Yaskawa INFORM job: X2_8A-21A(90,0)_DOD_WZM_BOK.JBI

/JOB
//NAME X2_8A-21A(90,0)_DOD_WZM_BOK
///FOLDERNAME X2
//POS
///NPOS 1047,1047,1047,43,0,0
///TOOL 0
///POSTYPE PULSE
///PULSE
C00000=-12667,-135547,-130714,31270,45596,0
C00001=-9315,-159766,-119262,-3212,6219,55552
C00002=-157761,-135547,-130714,31270,45596,-69143
C00003=-154472,-113934,-104337,41712,51336,-70449
C00004=-149832,-108771,-100172,39130,49259,-68869
C00005=-148058,-106656,-98467,38074,48499,-68236
C00006=-148062,-106275,-96666,38578,47777,-68578
C00007=-148058,-106656,-98467,38074,48499,-68236
C00008=-147997,-106381,-96958,38469,47847,-68508
C00009=-145894,-104035,-96109,36815,47477,-67498
C00010=-147997,-106381,-96958,38469,47847,-68508
C00011=-154410,-113635,-102825,42095,50721,-70729
C00012=-154342,-120637,-107041,25827,48602,-38771
C00013=-150292,-111683,-102360,22573,48994,-36710
C00014=-148798,-108210,-100464,21373,49171,-35962
C00015=-146664,-105787,-99597,19708,49308,-34937
C00016=-146949,-106220,-99797,19932,49282,-35074
C00017=-147721,-103636,-97533,20478,49410,-35405
C00018=-146949,-106220,-99797,19932,49282,-35074
C00019=-152261,-118724,-106469,24248,48548,-37770
C00020=-148295,-114597,-117137,-6490,60568,-69086
C00021=-147868,-109631,-111600,-6790,59752,-68875
C00022=-147704,-107727,-109395,-6911,59390,-68790
C00023=-147708,-107860,-107783,-6984,58336,-68724
C00024=-147704,-107727,-109395,-6911,59390,-68790
C00025=-147723,-107760,-107968,-6963,58499,-68740
C00026=-147306,-102596,-106094,-7098,60024,-68678
C00027=-147723,-107760,-107968,-6963,58499,-68740
C00028=-148315,-114751,-115749,-6537,59639,-69038
C00029=-148355,-114889,-117236,-6461,60467,-69101
C00030=-147925,-109892,-111692,-6763,59663,-68890
C00031=-147761,-107977,-109485,-6884,59305,-68805
C00032=-147764,-108104,-107870,-6957,58254,-68739
C00033=-147777,-108153,-108078,-6942,58354,-68751
C00034=-147358,-102980,-106206,-7078,59886,-68688
C00035=-147777,-108153,-108078,-6942,58354,-68751
C00036=-148373,-115211,-115873,-6515,59468,-69049
C00037=-147696,-122269,-111871,-35505,39043,-51945
C00038=-147690,-118447,-100224,-39719,34874,-49579
C00039=-148491,-109409,-94254,-38171,35277,-50420
C00040=-148787,-105724,-91002,-38010,35060,-50504
C00041=-148789,-105382,-89977,-38411,34697,-50285
C00042=-149058,-101689,-89016,-37046,35623,-51030
C00043=-149145,-100783,-88679,-36755,35795,-51189
C00044=-149058,-101689,-89016,-37046,35623,-51030
C00045=-145777,-99657,-88811,-39022,37803,-49998
C00046=-148139,-100407,-89095,-37251,36591,-50936
C00047=-145777,-99657,-88811,-39022,37803,-49998
C00048=-147690,-118447,-100224,-39719,34874,-49579
C00049=-128033,-128545,-103748,-39689,32513,-43973
C00050=-128383,-118409,-97778,-37905,33566,-44930
C00051=-128511,-114277,-94563,-37658,33626,-45064
C00052=-128512,-113804,-93446,-38069,33271,-44843
C00053=-129119,-111006,-93029,-36452,33958,-45715
C00054=-129434,-109852,-92636,-35862,34111,-46033
C00055=-128358,-113721,-93936,-37885,33613,-44941
C00056=-176216,-70111,-78093,55162,70856,-80763
C00057=-174311,-70781,-78417,54616,69674,-80426
C00058=-176216,-70111,-78093,55162,70856,-80763
C00059=-181747,-69996,-81392,56304,75271,-81045
C00060=-178033,-77165,-93769,42680,75059,-77098
C00061=-164745,-109340,-116699,-3009,62053,-68278
C00062=-145851,-112599,-102075,-47717,41998,-56322
C00063=-148044,-104803,-96379,-45883,41204,-57334
C00064=-148864,-101708,-93474,-45490,40644,-57533
C00065=-148866,-101457,-92299,-45986,40221,-57239
C00066=-148863,-101834,-94104,-45225,40876,-57690
C00067=-145127,-99228,-91361,-47944,42572,-56214
C00068=-147466,-100038,-91670,-46636,41186,-56907
C00069=-145127,-99228,-91361,-47944,42572,-56214
C00070=-146129,-107372,-95667,-48598,40993,-55782
C00071=-148216,-109089,-93488,-49289,38371,-55335
C00072=-148344,-107837,-93052,-48851,38553,-55585
C00073=-147906,-112054,-94498,-50363,37947,-54724
C00074=-145851,-112599,-102075,-47717,41998,-56322
C00075=-158250,-140903,-124067,-47621,67451,-49320
C00076=-161740,-133075,-117656,-46661,65672,-50232
C00077=-162335,-130592,-114553,-46699,64919,-50156
C00078=-162276,-129951,-113381,-46845,64676,-49998
C00079=-160420,-132544,-115533,-47350,65644,-49520
C00080=-135901,-74424,-73697,-74364,100921,-31256
C00081=-137788,-75503,-74147,-74218,99532,-31324
C00082=-138769,-76027,-74362,-74146,98812,-31363
C00083=-135901,-74424,-73697,-74364,100921,-31256
C00084=-149282,-147643,-98518,-79858,51263,-26133
C00085=-149394,-146891,-98381,-79629,51249,-26315
C00086=-148448,-152811,-99407,-81432,51428,-24854
C00087=-139735,-166147,-105854,-82069,56849,-22658
C00088=-180438,-97574,-115199,-33764,102267,52414
C00089=-189965,-108899,-115705,-31971,94091,51156
C00090=-190633,-110068,-115194,-31831,93066,51189
C00091=-190637,-110288,-114404,-31804,92551,51332
C00092=-190629,-109833,-115910,-31859,93547,51055
C00093=-186867,-102382,-113240,-32521,96788,51574
C00094=-187005,-102964,-110979,-32373,95300,51952
C00095=-188888,-106610,-112304,-32065,93703,51681
C00096=-187005,-102964,-110979,-32373,95300,51952
C00097=-188021,-107681,-112675,-32159,93748,52003
C00098=-189590,-103281,-111094,-32025,94271,51250
C00099=-188021,-107681,-112675,-32159,93748,52003
C00100=-180438,-97574,-115199,-33764,102267,52414
C00101=-185735,-83978,-109774,-33564,103394,50026
C00102=-199988,-77820,-108712,11582,98175,-38155
C00103=-204749,-56978,-92496,29836,109182,-47433
C00104=-202460,-56662,-91339,29422,107990,-46925
C00105=-201413,-57385,-91726,29256,107546,-46663
C00106=-201611,-57041,-91542,29296,107663,-46703
C00107=-201611,-58240,-90431,29070,106521,-47008
C00108=-203359,-50274,-87822,29763,109247,-46906
C00109=-195470,-25798,-72981,29209,109868,-43903
C00110=-195013,-27562,-73704,29036,109327,-43888
C00111=-194283,-28250,-74172,28893,109053,-43704
C00112=-194480,-28066,-74047,28932,109127,-43754
C00113=-194480,-29296,-73135,28708,108075,-44034
C00114=-195605,-24849,-71507,29147,109538,-44038
C00115=-191110,-5546,-57842,28597,109561,-42465
C00116=-192519,-3768,-54500,33008,111368,-41387
C00117=-191992,-5303,-55742,32912,111174,-41254
C00118=-192059,-5108,-55586,32924,111198,-41271
C00119=-192059,-6294,-54683,32651,110210,-41583
C00120=-192882,-2296,-53893,33162,111810,-41382
C00121=-203365,-15491,-64400,34648,115083,-44256
C00122=-218411,-26661,-75493,58573,107247,-46176
C00123=-145332,-87800,-123084,4045,108310,15756
C00124=-109199,-104290,-129101,-21867,105305,43874
C00125=-112610,-115777,-129409,-14908,94573,36374
C00126=-117115,-112620,-124614,-14006,92529,35127
C00127=-118008,-112320,-123068,-13816,91609,34934
C00128=-118007,-112900,-122267,-13806,90840,35020
C00129=-118044,-112536,-122505,-13803,91159,34973
C00130=-118576,-105776,-120168,-13731,93052,34586
C00131=-118044,-112536,-122505,-13803,91159,34973
C00132=-125955,-111499,-122045,-12179,90192,32457
C00133=-127333,-111877,-122174,-11884,89885,32033
C00134=-124755,-111115,-121914,-12435,90480,32824
C00135=-119624,-116552,-128230,-13509,92325,34321
C00136=-117231,-121833,-124467,-22052,85463,28755
C00137=-122341,-114124,-118662,-20866,84531,27121
C00138=-123318,-113111,-117155,-20643,83910,26885
C00139=-123641,-113323,-116249,-20585,83205,26892
C00140=-123595,-112804,-116375,-20585,83540,26851
C00141=-123397,-106736,-114247,-20589,85286,26623
C00142=-123595,-112804,-116375,-20585,83540,26851
C00143=-116023,-114044,-115764,-22346,84523,29358
C00144=-117346,-116777,-115957,-22098,82979,29171
C00145=-118867,-116723,-116143,-21757,82713,28674
C00146=-116293,-116772,-115815,-22329,83179,29512
C00147=-117231,-121833,-124467,-22052,85463,28755
C00148=-154726,-134692,-133300,19029,79240,32627
C00149=-155157,-123239,-125350,19102,80279,32639
C00150=-155214,-122106,-123677,19140,79867,32554
C00151=-155216,-122330,-122794,19175,79245,32454
C00152=-155272,-122641,-123186,19186,79334,32449
C00153=-154565,-115790,-120970,18882,81218,32994
C00154=-155272,-122449,-123985,19155,79894,32538
C00155=-110972,-119209,-121408,-15853,79302,48266
C00156=-109086,-133769,-122042,-16854,72857,49812
C00157=-111848,-135958,-122676,-16103,71595,48979
C00158=-109086,-133769,-122042,-16854,72857,49812
C00159=-108592,-130707,-130810,-16554,79646,49045
C00160=-120610,-122471,-119242,-21572,81234,22537
C00161=-120610,-122484,-118172,-21604,80613,22649
C00162=-120610,-122391,-116483,-21658,79689,22817
C00163=-120610,-122419,-116833,-21647,79876,22783
C00164=-120610,-122423,-116832,-21647,79874,22783
C00165=-120610,-122419,-116833,-21647,79876,22783
C00166=-120610,-122416,-116761,-21649,79836,22790
C00167=-120610,-122436,-116768,-21650,79830,22791
C00168=-120610,-122416,-116761,-21649,79836,22790
C00169=-120611,-122370,-120508,-21535,82009,22397
C00170=-120500,-119354,-126515,-17332,87675,17755
C00171=-155157,-123239,-125350,19102,80279,32639
C00172=-155214,-122106,-123677,19140,79867,32554
C00173=-155216,-122330,-122794,19175,79245,32454
C00174=-155272,-122641,-123186,19186,79334,32449
C00175=-154565,-115790,-120970,18882,81218,32994
C00176=-155272,-122449,-123985,19155,79894,32538
C00177=-110972,-119209,-121408,-15853,79302,48266
C00178=-109086,-133769,-122042,-16854,72857,49812
C00179=-111848,-135958,-122676,-16103,71595,48979
C00180=-109086,-133769,-122042,-16854,72857,49812
C00181=-108592,-130707,-130810,-16554,79646,49045
C00182=-120611,-118687,-129075,-3134,90000,4412
C00183=-120611,-121772,-123926,-3138,85252,4531
C00184=-120611,-122092,-122744,-3141,84362,4553
C00185=-120611,-122362,-121169,-3146,83256,4581
C00186=-120611,-122286,-121724,-3144,83636,4571
C00187=-120611,-122290,-121724,-3144,83633,4571
C00188=-120611,-122286,-121724,-3144,83636,4571
C00189=-120611,-121006,-125813,-3134,86805,4492
C00190=-120621,-113915,-131911,-13153,116790,34478
C00191=-136832,-143297,-133894,-19017,104291,40845
C00192=-187686,-122249,-118318,-34521,102174,42234
C00193=-187703,-122088,-115580,-34298,100833,42653
C00194=-187707,-122010,-114917,-34250,100525,42749
C00195=-187713,-121734,-113169,-34135,99743,42991
C00196=-187707,-122010,-114917,-34250,100525,42749
C00197=-187770,-121697,-112491,-32279,113674,44764
C00198=-187767,-121692,-112491,-32279,113678,44765
C00199=-187770,-121697,-112491,-32279,113674,44764
C00200=-187667,-121438,-112064,-34928,84963,41689
C00201=-187673,-121448,-112068,-34927,84958,41688
C00202=-187667,-121438,-112064,-34928,84963,41689
C00203=-187641,-121360,-124129,-34919,91154,39753
C00204=-178673,-119471,-127738,-23493,103847,53429
C00205=-160878,-120510,-126471,-37,121976,81968
C00206=-160881,-121699,-123664,-37,119637,81967
C00207=-160883,-121991,-122485,-37,118762,81967
C00208=-160886,-122244,-120905,-37,117660,81966
C00209=-160884,-122111,-121864,-37,118318,81967
C00210=-160882,-122100,-121862,-36,118322,81968
C00211=-160884,-122111,-121864,-37,118318,81967
C00212=-160879,-120821,-125908,-37,121469,81968
C00213=-160879,-120821,-131564,-37,121469,81968
C00214=-157394,-128671,-131753,738,117538,83283
C00215=-158801,-138021,-132727,409,113343,82737
C00216=-158801,-138035,-132347,409,113101,82737
C00217=-158801,-138034,-131509,408,112586,82736
C00218=-158801,-138039,-131833,408,112783,82736
C00219=-160693,-149427,-134985,6,108877,82039
C00220=-160612,-153549,-136083,24,107435,82069
C00221=-159125,-144348,-133603,336,110634,82611
C00222=-199963,-104116,-119881,11013,127404,83152
C00223=-204692,-116225,-118816,8637,121169,80600
C00224=-203581,-121519,-120530,8810,119404,80895
C00225=-204849,-113790,-122122,8953,124435,80816
C00226=-166129,-114439,-129167,13521,133132,-54375
C00227=-82387,-124374,-130385,21792,102809,-55833
C00228=-37550,-124758,-124791,27166,84975,-54517
C00229=-35933,-124831,-122904,26864,83389,-54284
C00230=-35589,-124875,-121597,26827,82538,-54351
C00231=-35584,-124889,-121174,26839,82296,-54405
C00232=-35764,-126387,-121953,26892,82093,-54519
C00233=-31633,-125451,-121673,25972,81076,-53208
C00234=-35764,-126387,-121953,26892,82093,-54519
C00235=-46981,-157328,-126723,35790,81436,-33730
C00236=-42905,-153934,-122174,35701,78867,-32870
C00237=-42758,-143813,-119569,35389,81762,-31868
C00238=-42905,-153934,-122174,35701,78867,-32870
C00239=-53188,-117519,-120731,36414,97747,-30962
C00240=-95179,-109851,-129540,3422,106316,17944
C00241=-143691,-100776,-119079,-26047,122130,73021
C00242=-146029,-112499,-120098,-24937,116556,73463
C00243=-147204,-116618,-119576,-24569,113992,73590
C00244=-147487,-116577,-118677,-24502,113425,73607
C00245=-146967,-116625,-120319,-24630,114475,73574
C00246=-147345,-121113,-121824,-24401,113105,73737
C00247=-146899,-128254,-123879,-23878,111030,74376
C00248=-147345,-121113,-121824,-24401,113105,73737
C00249=-118081,-135478,-120686,-30293,109901,65237
C00250=-118366,-136707,-118609,-29972,108136,65614
C00251=-120887,-140213,-119894,-30302,106351,65070
C00252=-118366,-136707,-118609,-29972,108136,65614
C00253=-117820,-130449,-123242,-31209,113594,64262
C00254=-93926,-103398,-125362,-18301,106221,39936
C00255=-72688,-110808,-124077,-7134,85250,24096
C00256=-75848,-101444,-116923,-6191,85411,23073
C00257=-76170,-100985,-115528,-6097,84767,23002
C00258=-76167,-101481,-114835,-6104,84090,23035
C00259=-78739,-96930,-113773,-5320,85595,22140
C00260=-79843,-95445,-113201,-4985,85938,21775
C00261=-77748,-98228,-114268,-5620,85298,22470
C00262=-140085,-104632,-109249,40944,98797,-6712
C00263=-140263,-103640,-106572,40817,98007,-7102
C00264=-137942,-102173,-106029,40697,97269,-6378
C00265=-140263,-103640,-106572,40817,98007,-7102
C00266=-135988,-101428,-112112,41019,99549,-4631
C00267=-141957,-83285,-117139,12315,91699,6710
C00268=-161957,-129781,-122866,-20018,67926,12328
C00269=-166016,-109699,-113650,-17211,72980,10098
C00270=-166795,-105246,-111748,-16434,74862,9605
C00271=-165677,-113012,-111900,-18316,68836,10778
C00272=-162725,-116093,-113629,-19548,69016,11850
C00273=-162651,-107484,-110669,-19284,71494,11460
C00274=-162725,-116093,-113629,-19548,69016,11850
C00275=-155151,-112727,-112486,-22270,71877,14160
C00276=-155120,-113819,-110277,-22518,70103,14518
C00277=-159000,-114269,-110433,-21107,68960,13264
C00278=-155120,-113819,-110277,-22518,70103,14518
C00279=-155137,-138999,-124748,-23105,66364,15269
C00280=-81055,-115973,-127517,23586,109336,-64560
C00281=-76492,-127739,-126040,22738,101683,-64421
C00282=-76072,-128597,-125529,22671,100870,-64425
C00283=-76065,-128640,-125326,22657,100732,-64448
C00284=-76072,-128576,-125785,22685,101025,-64394
C00285=-82641,-146978,-130130,22016,96499,-67668
C00286=-81130,-155003,-132256,21951,93476,-67670
C00287=-82641,-146978,-130130,22016,96499,-67668
C00288=-84000,-144678,-127518,21929,96467,-68175
C00289=-84000,-143983,-126065,21900,95967,-68269
C00290=-83327,-146231,-127404,21916,95478,-68108
C00291=-88356,-135439,-132684,22407,104994,-68175
C00292=-104080,-128245,-132212,-31995,84146,-22143
C00293=-106783,-105266,-117364,-31197,85468,-23533
C00294=-107129,-103609,-115494,-31111,85090,-23558
C00295=-107127,-104217,-114421,-31144,84251,-23329
C00296=-107044,-104571,-114816,-31164,84333,-23320
C00297=-107880,-99055,-112779,-30885,85404,-23924
C00298=-107044,-104571,-114816,-31164,84333,-23320
C00299=-105114,-115284,-123193,-31689,84721,-22698
C00300=-105208,-113465,-123990,-31624,85910,-23065
C00301=-106823,-104635,-117017,-31184,85549,-23570
C00302=-107122,-103295,-115264,-31113,85109,-23561
C00303=-107121,-103855,-114286,-31142,84342,-23351
C00304=-107087,-104437,-114776,-31151,84356,-23343
C00305=-107921,-98925,-112738,-30873,85426,-23945
C00306=-107087,-104437,-114776,-31151,84356,-23343
C00307=-105701,-116384,-125830,-31502,85418,-23114
C00308=-79137,-116524,-127291,-7118,77084,38210
C00309=-66518,-158449,-133200,-8588,59166,50817
C00310=-70166,-147728,-127011,-6864,60501,49298
C00311=-71549,-143558,-123868,-6244,60595,48757
C00312=-71544,-142942,-122687,-6271,60188,48782
C00313=-71412,-140542,-122600,-6259,61371,48766
C00314=-74130,-137647,-121783,-5023,62161,47690
C00315=-71412,-140542,-122600,-6259,61371,48766
C00316=-59221,-85077,-106862,-19044,97138,55247
C00317=-59772,-90133,-108950,-18878,95774,55276
C00318=-59221,-85077,-106862,-19044,97138,55247
C00319=-65406,-128676,-128270,-8670,80773,42177
C00320=-57064,-112054,-129147,-2862,108793,29097
C00321=-70948,-123089,-127271,10962,111372,-380
C00322=-67644,-116564,-123033,11394,111660,848
C00323=-67644,-116773,-122597,11361,111292,811
C00324=-67644,-116291,-123546,11437,112109,893
C00325=-70770,-123262,-125779,10903,110357,-412
C00326=-70770,-123588,-124717,10837,109552,-488
C00327=-69306,-120453,-123728,11077,110342,115
C00328=-70770,-123283,-125719,10898,110311,-416
C00329=-70770,-119886,-130778,11344,115083,53
C00330=-68413,-122856,-123349,22437,117236,58
C00331=-67404,-122631,-120786,22344,115611,123
C00332=-67401,-122683,-120099,22253,115193,37
C00333=-67283,-122594,-120333,22317,115338,115
C00334=-65261,-118175,-118917,23034,116088,1096
C00335=-67283,-122594,-120333,22317,115338,115
C00336=-70820,-123560,-126018,22187,119059,-540
C00337=-59587,-128850,-129971,-18356,103459,48793
C00338=-60648,-112549,-116046,-37363,97913,74718
C00339=-66648,-121539,-115269,-36526,91263,74498
C00340=-69624,-125916,-115212,-36242,88151,74300
C00341=-69624,-125773,-114639,-36242,87924,74374
C00342=-69624,-125814,-114800,-36242,87987,74354
C00343=-70738,-127677,-115368,-36152,87024,74211
C00344=-69624,-125814,-114800,-36242,87987,74354
C00345=-61556,-115340,-115782,-37136,96245,74919
C00346=-93863,-107857,-129738,-18786,98098,27923
C00347=-113340,-105978,-120535,-17383,92037,15860
C00348=-116256,-99504,-115214,-16745,91512,14962
C00349=-117355,-97038,-113094,-16498,91266,14630
C00350=-124053,-106600,-116618,-14934,87391,12894
C00351=-123019,-109757,-118902,-15179,87365,13243
C00352=-120254,-118381,-124729,-15823,87055,14212
C00353=-121076,-118719,-112405,-41381,81563,9211
C00354=-125328,-110839,-107644,-40465,80446,7775
C00355=-126920,-107772,-105722,-40091,80023,7243
C00356=-122279,-105715,-102241,-45382,81605,7865
C00357=-118123,-103314,-98388,-50429,83325,8212
C00358=-115452,-99808,-95169,-50805,84680,8860
C00359=-113598,-101964,-96694,-51043,85596,9323
C00360=-108732,-107177,-100380,-51565,88044,10518
C00361=-131658,-113091,-133069,-11905,90618,-13395
C00362=-155934,-143784,-122811,23124,58745,-32427
C00363=-151507,-132468,-117411,20635,59886,-30339
C00364=-149876,-128251,-115276,19729,60288,-29596
C00365=-151213,-128323,-114307,20456,60014,-30191
C00366=-146890,-120795,-114089,13688,65901,-25886
C00367=-142734,-111238,-112703,7950,73001,-22079
C00368=-143750,-114926,-115045,8343,72653,-22456
C00369=-146492,-125018,-121022,9420,71459,-23506
C00370=-146459,-122334,-129315,9145,77857,-23007
C00371=-118526,-115013,-133262,8809,105739,-46794
C00372=-93674,-118800,-129721,8134,120991,-68616
C00373=-93669,-120967,-127104,7892,118292,-68817
C00374=-94734,-125499,-127256,7488,116172,-69370
C00375=-102152,-150969,-134401,5465,108121,-72564
C00376=-93660,-121042,-127131,7893,118270,-68815
C00377=-93665,-118880,-129750,8134,120967,-68614
C00378=-98446,-113408,-116165,41475,93741,-73013
C00379=-95217,-118830,-115137,40946,89638,-73223
C00380=-92912,-120932,-114950,40678,87660,-72983
C00381=-96081,-129446,-114840,41081,85733,-75123
C00382=-96936,-125131,-114749,41104,87782,-74702
C00383=-101504,-121000,-116278,41571,92256,-74948
C00384=-100864,-122088,-112493,43204,76282,-71688
C00385=-96953,-122826,-110054,42689,72984,-71279
C00386=-94356,-123741,-109617,42253,71173,-70830
C00387=-94321,-123299,-107872,42432,70522,-71095
C00388=-95642,-121622,-108630,42447,72155,-71017
C00389=-100864,-121830,-111367,43291,75868,-71867
C00390=-131033,-115476,-133015,2815,101744,-74384
C00391=-151471,-119125,-123137,-34971,103386,-73225
C00392=-162012,-101235,-114016,-37763,108592,-75954
C00393=-165544,-104560,-113885,-37278,105688,-76399
C00394=-161186,-105898,-111701,-36934,105869,-74609
C00395=-157962,-101866,-111865,-37402,108959,-74341
C00396=-155898,-93647,-112180,-38609,113341,-75115
C00397=-93674,-112333,-133466,8753,126560,-68151
C00398=-93674,-118800,-129721,8134,120991,-68616
C00399=-93669,-120967,-127104,7892,118292,-68817
C00400=-93667,-121558,-126026,7814,117333,-68886
C00401=-93663,-121536,-126144,7822,117416,-68879
C00402=-93639,-121762,-126135,7818,117296,-68878
C00403=-93680,-121434,-126040,7817,117406,-68885
C00404=-93660,-121042,-127131,7893,118270,-68815
C00405=-93665,-118880,-129750,8134,120967,-68614
C00406=-98446,-113408,-116165,41475,93741,-73013
C00407=-93996,-117843,-114815,40802,89312,-72817
C00408=-91343,-117266,-113836,40455,87860,-72224
C00409=-92137,-119395,-114109,40564,87510,-72703
C00410=-95072,-126184,-113786,40951,86041,-74561
C00411=-95071,-125918,-112907,40977,85731,-74679
C00412=-96936,-125131,-114749,41104,87782,-74702
C00413=-101504,-121000,-116278,41571,92256,-74948
C00414=-100864,-122088,-112493,43204,76282,-71688
C00415=-95643,-121963,-109784,42340,72556,-70846
C00416=-93677,-120964,-108398,41948,71358,-70433
C00417=-93599,-120925,-107098,42100,70733,-70661
C00418=-95642,-121622,-108630,42447,72155,-71017
C00419=-100864,-121830,-111367,43291,75868,-71867
C00420=-131033,-115476,-133015,2815,101744,-74384
C00421=-151471,-119125,-123137,-34971,103386,-73225
C00422=-162012,-101235,-114016,-37763,108592,-75954
C00423=-163593,-104354,-113811,-37340,106547,-75879
C00424=-162938,-104376,-113793,-37349,106803,-75692
C00425=-158829,-104862,-111593,-37019,107224,-74083
C00426=-157962,-101866,-111865,-37402,108959,-74341
C00427=-155898,-93647,-112180,-38609,113341,-75115
C00428=-179206,-139250,-107986,-62075,77828,-66561
C00429=-185232,-138953,-105140,-62379,73225,-66913
C00430=-187696,-139015,-104542,-62453,71468,-67163
C00431=-187702,-137665,-102648,-62587,71237,-66963
C00432=-185238,-138055,-103864,-62461,73065,-66778
C00433=-179211,-138396,-106727,-62132,77661,-66424
C00434=-179188,-148562,-121526,-61524,79591,-68010
C00435=-184417,-115822,-131978,-19629,107310,7500
C00436=-190427,-134899,-136820,8574,116374,78562
C00437=-188066,-120573,-128029,9218,118052,79593
C00438=-191610,-147357,-136376,6897,103791,75181
C00439=-187795,-119828,-126345,9210,117376,79639
C00440=-187841,-121664,-124728,-2971,114560,78170
C00441=-187942,-121398,-126015,-3016,115485,78109
C00442=-187937,-119495,-128851,-3098,118205,78035
C00443=-176042,-128909,-129640,-7380,110692,58022
C00444=-187833,-113452,-115854,-34994,105139,41767
C00445=-187847,-113781,-113588,-34722,103839,42187
C00446=-187853,-113844,-112659,-34623,103335,42348
C00447=-187856,-113866,-111596,-34519,102780,42525
C00448=-187851,-113844,-112538,-34611,103274,42368
C00449=-187836,-113627,-114840,-34866,104547,41960
C00450=-186756,-108501,-120882,-36201,110201,40487
C00451=-150585,-129060,-123753,-46684,114085,-39870
C00452=-134046,-137019,-115206,-49635,112096,-74674
C00453=-134033,-140586,-110307,-48065,108843,-72866
C00454=-134037,-138671,-107458,-47843,108316,-72589
C00455=-133950,-137111,-106105,-47812,108341,-72556
C00456=-133930,-150358,-126108,1173,113974,-57522
C00457=-134040,-150029,-126001,1133,114079,-57562
C00458=-134505,-148512,-125722,2741,114238,-57140
C00459=-137673,-151162,-132623,1623,117206,-58299
C00460=-106012,-107394,-121753,14018,130776,-44816
C00461=-106669,-102485,-112824,13121,127987,-45519
C00462=-97512,-96218,-110425,14566,129183,-82759
C00463=-98864,-105619,-112306,13303,125832,-83842
C00464=-106150,-109468,-113796,12766,125107,-45727
C00465=-105474,-116823,-114648,29161,97726,-33837
C00466=-134074,-146851,-118858,40485,90771,-46834
C00467=-141855,-151854,-132376,33568,89282,-32323
C00468=-173958,-148748,-133240,11874,65312,15203
C00469=-187653,-128002,-123664,-7056,57779,46476
C00470=-188071,-112180,-99768,1790,31671,46486
C00471=-188092,-111455,-97340,1875,30550,46442
C00472=-187851,-111485,-96835,1581,30220,46589
C00473=-187792,-110201,-93997,1555,29133,46605
C00474=-187737,-110060,-93474,1490,28882,46636
C00475=-187785,-109075,-90961,1604,27844,46576
C00476=-188106,-109627,-92159,2030,28303,46362
C00477=-188086,-110531,-94662,1935,29378,46411
C00478=-188086,-114129,-114927,1479,39995,46659
C00479=-201470,-41376,-102585,19941,97743,-57993
C00480=-197439,-2624,-49840,39121,107911,-51008
C00481=-168348,92819,48556,27514,116832,-48709
C00482=-170146,82769,36005,28011,119675,-48673
C00483=-172466,59662,8523,30747,114377,-38085
C00484=-173361,44293,-8668,31536,116980,-37634
C00485=-173326,42548,-10417,31798,119739,-39927
C00486=-173293,31446,-22173,31559,124382,-42741
C00487=-170045,43132,-9775,28753,130915,-51393
C00488=-186843,33187,-28183,45340,118495,-56566
C00489=-187270,22965,-40018,42118,113549,-44205
C00490=-164927,12374,-50848,37497,97302,26684
C00491=-160848,-52651,-98971,6904,73590,44156
C00492=-187933,-111679,-98706,-278,30585,46526
C00493=-187953,-110958,-96368,-260,29517,46517
C00494=-188171,-110591,-95666,34,29272,46369
C00495=-188111,-109885,-93130,-50,28074,46412
C00496=-188090,-109778,-92606,-82,27808,46427
C00497=-188055,-108797,-90194,-133,26826,46455
C00498=-187968,-109087,-91174,-258,27282,46516
C00499=-187948,-109974,-93584,-278,28309,46526
C00500=-190713,-138118,-122139,3147,45685,54861
C00501=-188097,-104568,-127563,3199,90457,72619
C00502=-188112,-108983,-124849,3203,86524,72515
C00503=-196049,-130715,-128058,11352,73875,69900
C00504=-193131,-119078,-125609,7963,80164,71095
C00505=-187364,-124777,-127140,2732,76642,72458
C00506=-191510,-130298,-128202,6704,73471,71168
C00507=-188153,-109076,-124888,3215,86502,72501
C00508=-188138,-104664,-127604,3212,90434,72606
C00509=-187898,-111965,-120493,-16766,69565,69566
C00510=-187918,-113285,-117348,-17044,67055,69927
C00511=-188336,-115132,-116370,-17036,65483,70009
C00512=-188181,-112945,-115606,-17029,66143,69965
C00513=-188166,-113080,-115592,-17048,66072,69982
C00514=-187991,-112297,-115306,-17102,66325,70009
C00515=-187944,-113344,-117352,-17035,67023,69922
C00516=-187924,-112030,-120500,-16757,69531,69561
C00517=-180038,-109975,-126789,-2440,82512,-7441
C00518=-174468,-102021,-118148,-1871,82653,-17547
C00519=-174479,-103807,-115834,-1877,80312,-17516
C00520=-175021,-104384,-114967,-1695,79470,-17680
C00521=-174783,-104250,-115053,-1777,79597,-17606
C00522=-174170,-106690,-109656,-11758,69864,-18312
C00523=-172833,-107431,-109671,-12341,69693,-17819
C00524=-174390,-105691,-110273,-11607,70709,-18474
C00525=-174377,-104937,-112785,-11492,72607,-18653
C00526=-190845,-100837,-124447,13698,93294,-33124
C00527=-206306,-116062,-120388,37359,88631,-50073
C00528=-215039,-120395,-106715,50971,83253,-62053
C00529=-215038,-119729,-104733,51036,82687,-62365
C00530=-215037,-119445,-103934,51064,82464,-62488
C00531=-215047,-118488,-101366,51160,81769,-62880
C00532=-215047,-118800,-102176,51129,81987,-62759
C00533=-215049,-119543,-104187,51057,82539,-62453
C00534=-215012,-122438,-115563,50746,86080,-60488
C00535=-160845,-113405,-113287,47121,77099,31472
C00536=-160851,-113463,-110064,47446,75709,30781
C00537=-161282,-114943,-109409,47754,75135,30277
C00538=-161254,-114846,-109376,47745,75139,30294
C00539=-160788,-113231,-109982,47419,75724,30819
C00540=-160782,-112987,-114684,46949,77813,31850
C00541=-161690,-87231,-108001,36248,90547,80444
C00542=-156210,-91223,-102127,34873,83736,80390
C00543=-152348,-73560,-94415,33644,85868,82536
C00544=-158330,-83683,-104653,35339,89043,81248
C00545=-160758,-112853,-114863,36163,82877,78288
C00546=-160760,-113152,-111426,36317,81029,77674
C00547=-159491,-108015,-113138,31549,97627,78488
C00548=-160662,-113202,-114930,31505,96709,77777
C00549=-163626,-124672,-119545,29271,98661,76908
C00550=-164622,-129006,-121133,28240,99357,76613
C00551=-160757,-112482,-116558,30024,102576,77779
C00552=-160755,-111254,-119690,30396,104801,78387
C00553=-139139,-104942,-132434,5076,105021,81413
C00554=-120610,-140892,-128239,-26796,83300,73925
C00555=-124485,-139346,-124335,-26282,80622,73071
C00556=-128794,-174695,-130569,-28116,58521,76693
C00557=-123854,-173705,-127920,-33486,56775,79744
C00558=-127596,-155142,-123084,-28725,56836,77726
C00559=-128095,-155529,-122172,-29132,53686,78388
C00560=-128860,-155984,-126780,-25446,58633,74277
C00561=-138109,-135032,-133743,-8289,74304,51513
C00562=-203654,-125968,-124215,37381,73551,-30645
C00563=-201127,-103516,-110680,20461,62884,-59060
C00564=-201138,-104157,-107983,20829,61019,-59420
C00565=-201193,-104400,-106652,21043,60147,-59612
C00566=-201232,-104446,-106694,21063,60161,-59627
C00567=-200873,-105228,-106882,20926,59802,-59552
C00568=-201116,-104130,-107973,20816,61021,-59411
C00569=-201105,-103488,-110669,20449,62886,-59051
C00570=-198523,-119273,-121454,24683,77158,-64296
C00571=-174403,-100049,-121231,21877,99309,-62114
C00572=-174406,-102879,-118773,21681,96545,-62622
C00573=-172958,-103152,-117900,21399,95556,-62302
C00574=-174224,-104881,-115910,21520,93897,-63036
C00575=-174418,-104205,-117181,21599,94999,-62906
C00576=-174415,-101880,-119808,21752,97619,-62429
C00577=-185776,-93152,-118465,-1785,83350,-67432
C00578=-169060,-142396,-123848,-37084,49654,-60484
C00579=-174230,-113472,-108308,-34615,49911,-64397
C00580=-174247,-112967,-104740,-35556,48304,-63744
C00581=-174471,-112928,-103062,-35946,47380,-63468
C00582=-174489,-112275,-102294,-36008,47261,-63425
C00583=-174590,-112153,-101603,-36140,46922,-63333
C00584=-174396,-113097,-100663,-36857,46141,-62871
C00585=-174330,-114043,-100633,-37190,45762,-62656
C00586=-174129,-122060,-98220,-45554,37107,-60115
C00587=-174246,-112406,-102200,-36228,47262,-63291
C00588=-174229,-113129,-105847,-35265,48804,-63944
C00589=-182962,-136134,-123657,-29797,44727,-67038
C00590=-203654,-125968,-124215,37381,73551,-30645
C00591=-201127,-103516,-110680,20461,62884,-59060
C00592=-201138,-104157,-107983,20829,61019,-59420
C00593=-201193,-104400,-106652,21043,60147,-59612
C00594=-201232,-104446,-106694,21063,60161,-59627
C00595=-200873,-105228,-106882,20926,59802,-59552
C00596=-201116,-104130,-107973,20816,61021,-59411
C00597=-201105,-103488,-110669,20449,62886,-59051
C00598=-198523,-119273,-121454,24683,77158,-64296
C00599=-174403,-100049,-121231,21877,99309,-62114
C00600=-174406,-102879,-118773,21681,96545,-62622
C00601=-172958,-103152,-117900,21399,95556,-62302
C00602=-174224,-104881,-115910,21520,93897,-63036
C00603=-174418,-104205,-117181,21599,94999,-62906
C00604=-174415,-101880,-119808,21752,97619,-62429
C00605=-185776,-93152,-118465,-1785,83350,-67432
C00606=-169060,-142396,-123848,-37084,49654,-60484
C00607=-174230,-113472,-108308,-34615,49911,-64397
C00608=-174247,-112967,-104740,-35556,48304,-63744
C00609=-174471,-112928,-103062,-35946,47380,-63468
C00610=-174489,-112275,-102294,-36008,47261,-63425
C00611=-174590,-112153,-101603,-36140,46922,-63333
C00612=-174396,-113097,-100663,-36857,46141,-62871
C00613=-174330,-114043,-100633,-37190,45762,-62656
C00614=-174129,-122060,-98220,-45554,37107,-60115
C00615=-174246,-112406,-102200,-36228,47262,-63291
C00616=-175798,-117006,-109100,-34199,48210,-64559
C00617=-178617,-124532,-114828,-32467,46840,-65534
C00618=-210827,-121899,-127370,-35396,86436,-76908
C00619=-214505,-124636,-123608,-35577,86411,-76994
C00620=-214521,-124823,-120077,-35640,84542,-76397
C00621=-209595,-138372,-118962,-40572,76618,-76704
C00622=-215572,-134536,-117924,-37557,71164,-81051
C00623=-214545,-124844,-120083,-35636,84527,-76402
C00624=-214528,-124659,-123615,-35573,86395,-76999
C00625=-214596,-124890,-121786,-39550,96156,-78039
C00626=-214607,-124784,-118461,-39383,94595,-77461
C00627=-215336,-122839,-115954,-39308,93846,-77495
C00628=-215216,-123286,-113688,-39218,92622,-76995
C00629=-214785,-119888,-114308,-39371,94481,-77497
C00630=-214619,-124823,-118761,-39395,94718,-77513
C00631=-214540,-124430,-116246,-48349,86426,-68042
C00632=-214499,-123956,-126099,-48385,90728,-70182
C00633=-158797,-145907,-128305,-56145,74291,-56792
C00634=-118138,-117595,-113507,-59219,64127,-52420
C00635=-134091,-119062,-102284,-58108,50235,-52331
C00636=-134095,-117716,-98836,-59129,49460,-51612
C00637=-134657,-117185,-97454,-59366,48806,-51448
C00638=-134083,-121591,-110246,-11584,43366,-62365
C00639=-133895,-121523,-110170,-11744,43379,-62274
C00640=-133843,-121378,-109751,-11603,42967,-62923
C00641=-134088,-120272,-105685,-8075,39028,-71413
C00642=-134097,-120880,-107281,-7954,39689,-71484
C00643=-133538,-122024,-122159,-7272,48238,-71950
C00644=-134045,-120979,-109361,-39707,45136,-55893
C00645=-134048,-117179,-98466,-43015,41514,-53843
C00646=-133905,-117568,-98535,-40781,40764,-54269
C00647=-134181,-118830,-102497,-12918,37668,-61575
C00648=-134198,-119226,-102647,-12934,37556,-61565
C00649=-158314,-116202,-98556,34083,40870,-74489
C00650=-162364,-123197,-107171,35832,43944,-75497
C00651=-134045,-120979,-109361,-39707,45136,-55893
C00652=-132003,-121638,-109572,-41117,45917,-55073
C00653=-131002,-106489,-98392,-41164,47077,-55091
C00654=-131123,-103588,-88252,-50265,40796,-51296
C00655=-163242,-98975,-95762,18008,45953,-74760
C00656=-153405,-104865,-97946,10266,42608,-70493
C00657=-134148,-119761,-102793,-13034,37388,-61506
C00658=-126986,-126229,-93303,56145,28917,-85918
C00659=-131099,-132353,-104040,54087,33374,-85008
C00660=-133651,-114033,-99266,51853,45977,-77066
C00661=-134816,-132236,-131789,-6177,48808,-72548
C00662=-152519,-98596,-126841,-17039,86437,-59409
C00663=-167034,-82548,-116958,-26153,108191,-47353
C00664=-167227,-85698,-113927,-25595,104988,-46679
C00665=-154754,-79329,-105712,-37422,108521,-45283
C00666=-159285,-74428,-103512,-37136,107681,-46815
C00667=-167896,-62467,-97746,-36329,106502,-49789
C00668=-170836,-57718,-95291,-35960,106173,-50801
C00669=-180979,-58723,-101497,-23976,107062,-51805
C00670=-180909,-54943,-104050,-24554,110296,-52487
C00671=-168157,-75412,-102271,-33648,91006,-21456
C00672=-174012,-67106,-91297,-33471,82630,-14810
C00673=-175466,-61382,-85667,-32996,81659,-15067
C00674=-176013,-59150,-83405,-32819,81253,-15153
C00675=-202608,-62025,-89962,4221,78254,-36710
C00676=-159972,-87195,-101610,-14286,75081,-22762
C00677=-154310,-93015,-102157,-19304,70769,-24486
C00678=-154362,-96202,-104591,-19297,70625,-24481
C00679=-154503,-104813,-110762,-19306,69999,-24428
C00680=-155575,-73729,-96860,-32555,86012,-14938
C00681=-157088,-68154,-91284,-32096,84992,-15206
C00682=-157731,-66276,-89193,-31903,84490,-15302
C00683=-176839,-77218,-97385,-7105,75561,-28432
C00684=-165473,-80321,-98709,-11948,76053,-24715
C00685=-199796,-81518,-91231,35244,71315,-57262
C00686=-201423,-82172,-92479,35779,72324,-57601
C00687=-205660,-83542,-95477,37134,74990,-58446
C00688=-150225,-90058,-124320,-20069,81923,-14603
C00689=-88917,-116100,-126028,-29630,66347,39612
C00690=-48102,-114880,-112674,-35477,56596,75725
C00691=-53396,-105773,-101201,-33500,52497,74682
C00692=-53385,-105323,-98106,-34230,51099,75219
C00693=-48465,-101460,-95464,-40425,56724,79171
C00694=-72122,-108844,-98440,461,39847,55622
C00695=-53363,-105522,-99057,-19217,46878,60217
C00696=-53371,-105892,-101942,-18746,48378,59901
C00697=-53322,-113038,-104699,812,43724,42660
C00698=-53318,-112442,-102021,830,42382,42650
C00699=-53317,-112163,-100935,837,41857,42645
C00700=-53253,-112229,-97736,1547,37461,42516
C00701=-53300,-111445,-98358,1568,38246,42506
C00702=-51520,-115460,-104005,-179,39644,43460
C00703=-55761,-139961,-122674,-27476,66843,55729
C00704=-53542,-121644,-113892,-40363,83761,61539
C00705=-53523,-121175,-111327,-40444,82737,61941
C00706=-53533,-120846,-110023,-41635,87424,59647
C00707=-53533,-120798,-109834,-41636,87355,59676
C00708=-53529,-120315,-108043,-41648,86710,59935
C00709=-53536,-120580,-109029,-41640,87063,59791
C00710=-53556,-121151,-111460,-41628,87965,59422
C00711=-52633,-122748,-126719,-40391,89833,59612
C00712=-140119,-108661,-130674,-21165,82789,-25459
C00713=-161125,-123349,-120158,-18581,66270,-46079
C00714=-161135,-123185,-116439,-18891,64175,-45732
C00715=-161140,-122976,-114905,-19018,63381,-45597
C00716=-161216,-123269,-115002,-18998,63277,-45609
C00717=-162856,-121662,-114495,-18189,63396,-46272
C00718=-161212,-123488,-116538,-18871,64068,-45743
C00719=-161202,-123677,-120265,-18562,66156,-46089
C00720=-167124,-146469,-125858,32695,63076,-70922
C00721=-161220,-122264,-110536,44525,64077,-74742
C00722=-161219,-121375,-107584,44985,63095,-75224
C00723=-164956,-113855,-102560,48427,66781,-75111
C00724=-161213,-120936,-106323,43985,60856,-74418
C00725=-161480,-119492,-104017,44742,56174,-74995
C00726=-161477,-119788,-101535,47560,52624,-77093
C00727=-161197,-119682,-102993,46927,53134,-76618
C00728=-161197,-120736,-105876,46275,53998,-76117
C00729=-161177,-121556,-108554,35078,57327,-43050
C00730=-161177,-120932,-106617,35398,56609,-43319
C00731=-152937,-127654,-109782,25136,48983,-42100
C00732=-161176,-119640,-103030,36318,54707,-44163
C00733=-161179,-121241,-107541,34339,64662,-45277
C00734=-161179,-121533,-108462,34233,65010,-45160
C00735=-161180,-122193,-110741,33972,65899,-44866
C00736=-159909,-111206,-128347,-10927,59798,-43136
C00737=-174276,-119239,-128019,9099,73009,32604
C00738=-174287,-122281,-118814,9519,65873,32039
C00739=-174304,-122135,-115653,9666,64029,31878
C00740=-174310,-121974,-114355,9727,63324,31815
C00741=-174277,-122172,-120616,-9764,82080,37769
C00742=-174277,-122177,-120568,-9764,82048,37772
C00743=-174317,-121775,-113110,-33515,107538,43031
C00744=-174312,-121937,-114098,-33622,107981,42892
C00745=-174299,-122214,-116525,-33911,109120,42531
C00746=-174287,-119835,-127268,-36019,115609,40290
C00747=-174287,-120021,-127206,9145,72119,32532
C00748=-174287,-120021,-127206,9145,72119,32532
C00749=-173736,-117333,-114872,9262,65925,32245
C00750=-174960,-111711,-111152,9771,66659,31859
C00751=-176831,-126585,-121826,-8311,79476,36809
C00752=-157010,-133467,-117360,-32643,99223,56368
C00753=-154345,-130153,-124672,-33336,105500,55567
C00754=-146682,-141770,-131473,-27794,101884,56245
C00755=-146682,-141770,-131473,-27794,101884,56245
C00756=-146682,-141770,-131473,15257,98468,53705
C00757=-102938,-141770,-131473,49664,98468,53705
C00758=-102938,-145417,-131473,49512,65454,53705
C00759=-103656,-129714,-109721,51674,62395,51470
C00760=-102995,-138917,-102303,63406,51064,43511
C00761=-104839,-135559,-111699,50177,75701,60454
C00762=-99828,-171084,-120161,53403,64595,56658
C00763=-110163,-126067,-103455,56717,91063,66073
C00764=-116435,-131456,-112749,56730,96510,65994
C00765=-116383,-133294,-113279,56655,96128,65766
C00766=-84454,-125099,-129012,35107,90636,33075
C00767=-15972,-110889,-128286,-10965,59905,-43045
C00768=-15972,-110889,-128286,-10965,59905,-43045
C00769=-53465,-86935,-89811,-40465,79071,68727
C00770=-108812,15435,-43443,-8262,104585,64007
C00771=-120685,104729,62045,12414,91835,74489
C00772=-120504,102152,62779,12366,90072,74374
C00773=-120431,101212,63194,12350,89339,74325
C00774=-120431,101002,64582,12347,88398,74232
C00775=-120431,101212,63194,12350,89339,74325
C00776=-121076,107244,72775,12456,86702,73844
C00777=-120665,102968,67176,12385,87860,74099
C00778=-121076,107244,72775,12456,86702,73844
C00779=-121323,110426,71256,12493,89251,74016
C00780=-131278,69881,50181,9127,63188,62805
C00781=-131485,74883,60411,9547,59533,62414
C00782=-131548,76399,63510,9674,58426,62296
C00783=-131548,76704,64506,9721,57977,62255
C00784=-131183,71204,57206,9397,59578,62541
C00785=-131068,71487,58412,9405,58972,62536
C00786=-131266,74091,61533,9552,58423,62408
C00787=-131382,69379,53589,9372,60872,62574
C00788=-130781,63634,40058,8705,66118,63219
C00789=-132526,40318,17232,-3897,63337,79864
C00790=-132770,43850,25861,-3900,59836,79894
C00791=-132775,45020,27808,-3921,59239,79913
C00792=-132775,45119,28557,-3937,58830,79928
C00793=-131974,40901,23457,-4303,59840,80201
C00794=-131974,41007,24367,-4325,59336,80221
C00795=-132343,43569,27070,-4148,58978,80090
C00796=-132425,41720,24361,-4076,59689,80031
C00797=-131916,36045,14544,-4216,62827,80109
C00798=-154350,3292,-38754,752,86522,75713
C00799=-181553,89062,52820,1715,95022,75090
C00800=-181735,85640,53357,1725,92938,75001
C00801=-181765,85113,53499,1727,92580,74986
C00802=-181767,85098,55139,1725,91564,74972
C00803=-181765,85113,53499,1727,92580,74986
C00804=-181351,93067,65191,1686,89465,75083
C00805=-181572,88775,59771,1706,90599,75024
C00806=-181351,93067,65191,1686,89465,75083
C00807=-181147,96755,64289,1671,91909,75184
C00808=-159394,22511,-602,-1012,64107,82504
C00809=-159231,25736,7387,-1125,60850,82595
C00810=-159081,26911,9255,-1209,60307,82658
C00811=-159081,26976,10155,-1214,59786,82663
C00812=-159081,26911,9255,-1209,60307,82658
C00813=-159295,23244,6238,-1098,60277,82577
C00814=-159295,23278,6733,-1101,59990,82580
C00815=-159347,25129,8513,-1077,59844,82563
C00816=-159295,23278,6733,-1101,59990,82580
C00817=-159427,17860,-3265,-1001,63356,82499
C00818=-180998,44453,11386,9428,69103,75000
C00819=-180806,46143,18147,9552,65832,74803
C00820=-180780,46418,19112,9573,65382,74775
C00821=-180783,46335,20682,9650,64387,74690
C00822=-180780,46418,19112,9573,65382,74775
C00823=-181199,40700,14756,9793,65178,74604
C00824=-180944,43672,17889,9700,64752,74662
C00825=-181199,40700,14756,9793,65178,74604
C00826=-181427,38720,7071,9647,68865,74830
C00827=-152316,-9212,-39627,-4041,74028,47424
C00828=-97675,-116344,-75406,-30929,43249,-3453
C00829=-144147,-96317,-43020,16665,22045,18189
C00830=-130185,-5552,7433,-2044,36537,82607
C00831=-148170,9866,-4864,-2727,74191,81047
C00832=-160677,16615,-6140,-3325,93789,80088
C00833=-160892,14618,-3978,-3294,91428,80078
C00834=-160979,13901,-3035,-3283,90476,80074
C00835=-160981,13982,-1301,-3281,89453,80100
C00836=-160979,13901,-3035,-3283,90476,80074
C00837=-160903,19705,2788,-3289,89879,80114
C00838=-160903,19733,3315,-3289,89569,80123
C00839=-160898,16854,1424,-3289,89254,80133
C00840=-160903,19794,4169,-3288,89076,80136
C00841=-160610,22295,943,-3323,92353,80148
C00842=-159769,-26352,-42847,7626,75430,42908
C00843=-160661,-23608,-37245,8003,73495,42476
C00844=-160801,-19429,-32426,8083,72699,42375
C00845=-160801,-19408,-31304,8110,72027,42329
C00846=-161009,-22449,-34949,8156,72720,42303
C00847=-161249,-23550,-34138,8284,71688,42148
C00848=-161035,-21507,-32672,8205,71812,42231
C00849=-161249,-23550,-34138,8284,71688,42148
C00850=-159612,-30937,-44211,7622,73912,42867
C00851=-144117,-44081,-61004,-17211,89666,8724
C00852=-145648,-40124,-55468,-16926,88039,8426
C00853=-146237,-38515,-53215,-16819,87384,8313
C00854=-146244,-38444,-53170,-16818,87391,8310
C00855=-146245,-38577,-51594,-16825,86395,8446
C00856=-146244,-38444,-53170,-16818,87391,8310
C00857=-146240,-38608,-52193,-16823,86734,8401
C00858=-146535,-35573,-50236,-16765,87015,8261
C00859=-146268,-38521,-51765,-16819,86519,8421
C00860=-147801,-39090,-52130,-16535,86146,7942
C00861=-146268,-38521,-51765,-16819,86519,8421
C00862=-144117,-44081,-61004,-17211,89666,8724
C00863=-145162,-56828,-95851,-3587,97052,36303
C00864=-147136,-55674,-91646,-3015,94990,35768
C00865=-150906,-56103,-90461,-1950,93937,34650
C00866=-150909,-57277,-89363,-1945,92659,34669
C00867=-150906,-56103,-90461,-1950,93937,34650
C00868=-147900,-55107,-89916,-2796,94193,35556
C00869=-147871,-56692,-89008,-2798,92822,35595
C00870=-149697,-57326,-89351,-2285,92656,35040
C00871=-147871,-56692,-89008,-2798,92822,35595
C00872=-149264,-52275,-86592,-2410,93564,35155
C00873=-149536,-48545,-84471,-2336,94168,35061
C00874=-149264,-52275,-86592,-2410,93564,35155
C00875=-145162,-56828,-95851,-3587,97052,36303
C00876=-148725,-41791,-46801,-46253,72923,-63254
C00877=-150766,-40622,-42529,-46203,70442,-63063
C00878=-151577,-40068,-40761,-46203,69457,-62988
C00879=-152585,-23504,-29643,-45527,70124,-63820
C00880=-151861,-23991,-31407,-45521,71087,-63922
C00881=-150038,-24992,-35653,-45558,73508,-64179
C00882=-157424,-58492,-62688,-32217,54755,-56547
C00883=-158288,-54308,-56839,-32290,53193,-56420
C00884=-158489,-51803,-54002,-32356,52725,-56354
C00885=-162920,-52118,-54243,-29783,51091,-57961
C00886=-162018,-54402,-56899,-30142,51809,-57760
C00887=-161259,-58664,-62788,-30049,53328,-57890
C00888=-162071,-38381,-52824,-22779,71448,-67723
C00889=-163630,41,-22976,-9730,99876,-85306
C00890=-164211,-2681,-21394,-9632,97468,-85315
C00891=-164465,-2984,-20111,-9597,96504,-85326
C00892=-167232,-2580,-19786,-9490,96192,-86245
C00893=-166888,-2331,-21114,-9528,97164,-86203
C00894=-166273,343,-22730,-9627,99573,-86181
C00895=-147061,-19099,-23009,-3757,61390,-3418
C00896=-130185,-5552,7433,-2044,36537,20417
C00897=-144147,-96317,-43020,16665,22045,18189
C00898=-97675,-116344,-75406,-30929,43249,-3453
C00899=-152316,-9212,-39627,-4041,74028,-36586
C00900=-151393,-4993,-15312,-4384,44467,-75506
C00901=-149831,-2435,-10935,-5835,43191,-74682
C00902=-153598,-2863,-5088,4597,34036,-78104
C00903=-153144,-5743,-2041,16094,25401,-81582
C00904=-154914,-1885,-10222,12324,42496,-79899
C00905=-154718,-4280,-13376,11999,43163,-79709
C00906=-167718,15574,1984,-24206,55458,-53961
C00907=-167855,19598,9384,-24857,53146,-53442
C00908=-167909,21312,12472,-25150,52202,-53220
C00909=-169559,21751,12884,-24222,51683,-53852
C00910=-169779,21817,12946,-24097,51615,-53936
C00911=-170327,21990,13109,-23783,51447,-54148
C00912=-170290,20267,10006,-23488,52399,-54367
C00913=-170195,16223,2573,-22831,54729,-54878
C00914=-178256,99378,67031,-19051,88552,-69176
C00915=-178526,97657,68868,-19024,86580,-68963
C00916=-178635,97078,69748,-19021,85760,-68874
C00917=-179853,98823,71988,-18874,85023,-69192
C00918=-179980,99017,72237,-18859,84943,-69225
C00919=-180384,99643,73043,-18810,84684,-69328
C00920=-180272,100173,72105,-18809,85516,-69417
C00921=-179996,101790,70145,-18825,87512,-69628
C00922=-171488,21123,-18735,-439,89529,-9365
C00923=-148539,8283,-18518,11481,74800,46031
C00924=-133884,78471,30098,11624,77529,65496
C00925=-133939,79564,34318,11736,75541,65288
C00926=-133726,80326,36877,11703,74352,65242
C00927=-129986,86296,44341,10172,72375,66337
C00928=-130560,84597,41197,10369,73487,66234
C00929=-130480,83524,36335,10225,75880,66464
C00930=-133789,96970,48697,23463,95575,62558
C00931=-133554,94997,50328,23328,93653,62262
C00932=-133996,90156,45840,23419,94027,62179
C00933=-133380,91261,47236,23299,93592,62310
C00934=-133261,94504,51359,23246,92757,62189
C00935=-128474,99178,56254,18479,90935,62982
C00936=-126544,95607,50814,14280,92008,63224
C00937=-126033,96144,51503,14181,91777,63369
C00938=-125984,92855,44553,14229,94278,63672
C00939=-118409,86943,34254,-498,98079,29639
C00940=-113225,75702,29820,-12477,90617,28537
C00941=-112952,75485,30802,-12536,89960,28691
C00942=-117762,67578,21374,-3134,88425,17539
C00943=-120996,68894,22851,4133,88343,9509
C00944=-120986,83403,30534,4203,100743,9917
C00945=-131138,87625,41047,12528,91017,-11277
C00946=-131518,88313,46232,13974,85364,-12988
C00947=-131574,88042,47103,13998,84717,-13081
C00948=-131699,87452,47047,14037,84474,-13150
C00949=-127523,76387,33616,3918,83280,-1876
C00950=-130224,83461,42270,11062,83726,-9611
C00951=-130883,82631,32190,11215,89482,-9310
C00952=-138903,29280,-14444,28707,91021,50587
C00953=-152753,-113498,-70464,41238,43505,17390
C00954=-199062,-57325,-47228,38260,64183,4080
C00955=-144700,-70309,-53328,-41384,55522,-26317
C00956=-159027,-8981,-29340,-14833,99808,-55594
C00957=-158734,-10357,-26337,-14717,97386,-55198
C00958=-158565,-10606,-24902,-14680,96435,-55024
C00959=-156379,-10444,-24769,-14732,96828,-54309
C00960=-156533,-10130,-26155,-14772,97783,-54479
C00961=-156840,-8773,-29171,-14894,100200,-54881
C00962=-162486,-26662,-42491,-16083,70936,-60571
C00963=-162478,-24897,-37244,-16311,68704,-60258
C00964=-161179,-32593,-36996,-20221,58130,-58095
C00965=-158572,-32392,-36861,-21515,58809,-57144
C00966=-159367,-24765,-36916,-18592,69259,-59149
C00967=-159276,-26541,-42171,-18380,71485,-59471
C00968=-144700,-70309,-53328,-41384,55522,-26317
C00969=-199062,-57325,-47228,38260,64183,4080
C00970=-152753,-113498,-70464,41238,43505,17390
C00971=-138903,29280,-14444,28707,91021,50587
C00972=-134460,43790,22046,6339,61230,73811
C00973=-133863,45767,26803,6146,59285,73930
C00974=-134087,48465,31540,6362,57781,73758
C00975=-130025,54134,37725,4242,56630,75317
C00976=-129992,52392,35365,4200,57178,75352
C00977=-129939,49644,28351,4047,60072,75482
C00978=-131463,16549,-4479,-10803,54184,75739
C00979=-132193,19578,1957,-10644,51724,75694
C00980=-132626,21348,4069,-10405,51283,75555
C00981=-134889,19383,2337,-8835,51077,74604
C00982=-134234,16346,-1785,-9163,52111,74787
C00983=-134362,13693,-7099,-8856,53981,74568
C00984=-136755,-2244,-27091,-2141,60146,66966
C00985=-152753,-113498,-70464,41238,43505,17390
C00986=-199062,-57325,-47228,38260,64183,4080
C00987=-144700,-70309,-53328,-41384,55522,-26317
C00988=-155243,-37029,-47289,-14287,81392,-50093
C00989=-162013,-14853,-33688,2862,92831,-64763
C00990=-161094,-16180,-30749,2749,90312,-64514
C00991=-160723,-16617,-29501,2705,89308,-64411
C00992=-157149,-16390,-29322,2290,89205,-63218
C00993=-157529,-15990,-30598,2335,90205,-63327
C00994=-158470,-14757,-33607,2451,92716,-63592
C00995=-164755,-27863,-42732,4142,59506,-66566
C00996=-163775,-25128,-37158,3650,57439,-66261
C00997=-162063,-21722,-33626,2650,56947,-65603
C00998=-158969,-21729,-33662,803,56902,-64386
C00999=-159524,-25179,-37184,1127,57304,-64599
C01000=-160428,-28024,-42833,1630,59333,-64922
C01001=-144700,-70309,-53328,-41384,55522,-26317
C01002=-199062,-57325,-47228,38260,64183,4080
C01003=-152753,-113498,-70464,41238,43505,17390
C01004=-177120,62510,20627,9539,95868,-53949
C01005=-182918,102274,70865,2025,89904,-72285
C01006=-182573,99881,71746,1990,88125,-72198
C01007=-182434,99026,72237,1977,87381,-72163
C01008=-177980,92594,64030,1535,89029,-70642
C01009=-178132,93443,63515,1551,89785,-70684
C01010=-178509,95798,62536,1591,91604,-70787
C01011=-170148,25411,11260,-10861,54110,-56839
C01012=-169779,29504,18940,-11463,51585,-56403
C01013=-169678,31092,21995,-11696,50557,-56237
C01014=-164974,29903,20823,-14564,51428,-54281
C01015=-165316,28440,17904,-14160,52381,-54569
C01016=-165615,24318,10218,-13532,54869,-55036
C01017=-177120,62510,20627,9539,95868,-53949
C01018=-152753,-113498,-70464,41238,43505,17390
C01019=-199062,-57325,-47228,38260,64183,4080
C01020=-144700,-70309,-53328,-41384,55522,-26317
C01021=-142540,-54200,-62960,-20837,71495,-76935
C01022=-143745,-53250,-58469,-20670,69060,-76947
C01023=-143907,-52449,-56432,-20721,68229,-76859
C01024=-146015,-19661,-41212,-16744,94255,-78829
C01025=-145325,-27004,-46307,-16815,93781,-78527
C01026=-145058,-29561,-48130,-16841,93649,-78418
C01027=-144903,-28900,-49357,-16896,94730,-78514
C01028=-144163,-26309,-51550,-17103,97446,-78641
C01029=-174273,-50790,-66274,-423,45257,-81721
C01030=-174293,-46300,-60313,-415,43895,-81724
C01031=-174300,-44502,-57900,-412,43334,-81724
C01032=-174308,-44682,-54936,-420,41418,-81719
C01033=-174300,-46542,-57382,-423,41967,-81718
C01034=-174281,-51187,-63424,-430,43299,-81715
C01035=-170286,-21589,-54734,-4189,80944,-76248
C01036=-174005,35790,2399,-5860,112639,-83034
C01037=-174229,31517,1683,-5803,110877,-83024
C01038=-174320,29862,1474,-5782,110152,-83021
C01039=-174151,30232,3489,-5706,109139,-82910
C01040=-174234,31116,4346,-5726,109041,-82935
C01041=-174010,35219,4888,-5776,110822,-82944
C01042=-165073,-12180,-39998,-12766,95090,-81399
C01043=-146454,-66354,-59123,-37370,62542,-80053
C01044=-148014,-113391,-77231,-42747,49474,-76607
C01045=-120872,-104982,-67229,-50399,61266,-16237
C01046=-12667,-135547,-130714,31270,45596,0
BC00000=78393,670967,1075175
BC00001=177059,727519,1002542
BC00002=78393,913126,1075175
BC00003=70793,903989,1075175
BC00004=70793,903989,1075175
BC00005=70793,903989,1075175
BC00006=70793,903989,1075175
BC00007=70793,903989,1075175
BC00008=70793,903989,1075175
BC00009=70793,903989,1075175
BC00010=70793,903989,1075175
BC00011=70793,903989,1075175
BC00012=103901,897249,1075175
BC00013=103901,897249,1075175
BC00014=103901,897249,1075175
BC00015=103901,897249,1075175
BC00016=103901,897249,1075175
BC00017=103901,897249,1075175
BC00018=103901,897249,1075175
BC00019=103901,897249,1075175
BC00020=89915,910531,1075175
BC00021=89915,910531,1075175
BC00022=89915,910531,1075175
BC00023=89915,910531,1075175
BC00024=89915,910531,1075175
BC00025=89915,910531,1075175
BC00026=89915,910531,1075175
BC00027=89915,910531,1075175
BC00028=89915,910531,1075175
BC00029=27368,899646,1075175
BC00030=27368,899646,1075175
BC00031=27368,899646,1075175
BC00032=27368,899646,1075175
BC00033=27368,899646,1075175
BC00034=27368,899646,1075175
BC00035=27368,899646,1075175
BC00036=27368,899646,1075175
BC00037=160753,772187,1075175
BC00038=160753,772187,1075175
BC00039=160753,772187,1075175
BC00040=160753,772187,1075175
BC00041=160753,772187,1075175
BC00042=160753,772187,1075175
BC00043=160753,772187,1075175
BC00044=160753,772187,1075175
BC00045=160753,772187,1075175
BC00046=160753,772187,1075175
BC00047=160753,772187,1075175
BC00048=160753,772187,1075175
BC00049=123402,765716,1075175
BC00050=123402,765716,1075175
BC00051=123402,765716,1075175
BC00052=123402,765716,1075175
BC00053=123402,765716,1075175
BC00054=123402,765716,1075175
BC00055=123402,765716,1075175
BC00056=123402,765716,1075175
BC00057=123402,765716,1075175
BC00058=123402,765716,1075175
BC00059=123402,765716,1075175
BC00060=129464,768278,1075175
BC00061=151149,777443,1075175
BC00062=169689,785624,1075175
BC00063=169689,785624,1075175
BC00064=169689,785624,1075175
BC00065=169689,785624,1075175
BC00066=169689,785624,1075175
BC00067=169689,785624,1075175
BC00068=169689,785624,1075175
BC00069=169689,785624,1075175
BC00070=169689,785624,1075175
BC00071=169689,785624,1075175
BC00072=169689,785624,1075175
BC00073=169689,785624,1075175
BC00074=169689,785624,1075175
BC00075=120114,813651,1075175
BC00076=120114,813651,1075175
BC00077=120114,813651,1075175
BC00078=120114,813651,1075175
BC00079=120114,813651,1075175
BC00080=120114,813651,1075175
BC00081=120114,813651,1075175
BC00082=120114,813651,1075175
BC00083=120114,813651,1075175
BC00084=120114,813651,1075175
BC00085=120114,813651,1075175
BC00086=120114,813651,1075175
BC00087=120114,813651,1075175
BC00088=141881,838168,1075175
BC00089=141881,838168,1075175
BC00090=141881,838168,1075175
BC00091=141881,838168,1075175
BC00092=141881,838168,1075175
BC00093=141881,838168,1075175
BC00094=141881,838168,1075175
BC00095=141881,838168,1075175
BC00096=141881,838168,1075175
BC00097=141881,838168,1075175
BC00098=141881,838168,1075175
BC00099=141881,838168,1075175
BC00100=141881,838168,1075175
BC00101=69874,805894,1075175
BC00102=70019,750208,1075175
BC00103=70019,750208,1075175
BC00104=70019,750208,1075175
BC00105=70019,750208,1075175
BC00106=70019,750208,1075175
BC00107=70019,750208,1075175
BC00108=70019,750208,1075175
BC00109=70019,750208,1075175
BC00110=70019,750208,1075175
BC00111=70019,750208,1075175
BC00112=70019,750208,1075175
BC00113=70019,750208,1075175
BC00114=70019,750208,1075175
BC00115=70018,750208,1075172
BC00116=70018,750208,1075172
BC00117=70018,750208,1075172
BC00118=70018,750208,1075172
BC00119=70018,750208,1075172
BC00120=70018,750208,1075172
BC00121=70018,750208,1075172
BC00122=70018,750208,1075172
BC00123=110204,822960,1075174
BC00124=128430,855958,1075175
BC00125=125005,945340,1075175
BC00126=125005,945340,1075175
BC00127=125005,945340,1075175
BC00128=125005,945340,1075175
BC00129=125005,945340,1075175
BC00130=125005,945340,1075175
BC00131=125005,945340,1075175
BC00132=125005,945340,1075175
BC00133=125005,945340,1075175
BC00134=125005,945340,1075175
BC00135=125005,945340,1075175
BC00136=177748,940008,1075175
BC00137=177748,940008,1075175
BC00138=177748,940008,1075175
BC00139=177748,940008,1075175
BC00140=177748,940008,1075175
BC00141=177748,940008,1075175
BC00142=177748,940008,1075175
BC00143=177748,940008,1075175
BC00144=177748,940008,1075175
BC00145=177748,940008,1075175
BC00146=177748,940008,1075175
BC00147=177748,940008,1075175
BC00148=225975,953000,1075175
BC00149=225975,953000,1075175
BC00150=225975,953000,1075175
BC00151=225975,953000,1075175
BC00152=225975,953000,1075175
BC00153=225975,953000,1075175
BC00154=225975,953000,1075175
BC00155=225975,953000,1075175
BC00156=225975,953000,1075175
BC00157=225975,953000,1075175
BC00158=225975,953000,1075175
BC00159=225975,953000,1075175
BC00160=254413,953027,1075175
BC00161=252547,954523,1075175
BC00162=252548,954519,1075175
BC00163=252583,954651,1075175
BC00164=252019,957675,1075175
BC00165=252583,954651,1075175
BC00166=252165,954787,1075175
BC00167=249030,954243,1075175
BC00168=252165,954787,1075175
BC00169=258696,949550,1075175
BC00170=257059,950024,1075175
BC00171=265795,953000,1075175
BC00172=265795,953000,1075175
BC00173=265795,953000,1075175
BC00174=265795,953000,1075175
BC00175=265795,953000,1075175
BC00176=265795,953000,1075175
BC00177=265795,953000,1075175
BC00178=265795,953000,1075175
BC00179=265795,953000,1075175
BC00180=265795,953000,1075175
BC00181=265795,953000,1075175
BC00182=254634,951648,1075175
BC00183=253737,956448,1075175
BC00184=253378,958368,1075175
BC00185=253379,958364,1075175
BC00186=253259,958395,1075175
BC00187=252695,961419,1075175
BC00188=253259,958395,1075175
BC00189=254515,951675,1075175
BC00190=248439,993035,1075175
BC00191=271638,1017285,1075175
BC00192=314947,1062557,1075175
BC00193=311280,1056373,1075175
BC00194=310409,1054905,1075175
BC00195=310409,1054901,1075175
BC00196=310409,1054905,1075175
BC00197=284329,1066137,1075175
BC00198=285931,1063482,1075175
BC00199=284329,1066137,1075175
BC00200=333588,1039325,1075175
BC00201=330835,1037779,1075175
BC00202=333588,1039325,1075175
BC00203=340460,1045393,1075175
BC00204=319968,1046454,1075175
BC00205=279319,1048558,1075175
BC00206=281895,1044284,1075175
BC00207=282926,1042574,1075175
BC00208=282926,1042570,1075175
BC00209=282744,1042486,1075175
BC00210=284346,1039831,1075175
BC00211=282744,1042486,1075175
BC00212=279137,1048470,1075175
BC00213=253507,1028204,1074244
BC00214=253507,1028204,1074244
BC00215=253507,1028204,1074244
BC00216=253507,1028204,1074244
BC00217=253507,1028204,1074244
BC00218=253507,1028204,1074244
BC00219=253507,1028204,1074244
BC00220=253507,1028204,1074244
BC00221=253507,1028204,1074244
BC00222=253507,1028204,1074244
BC00223=253507,1028204,1074244
BC00224=253507,1028204,1074244
BC00225=253507,1028204,1074244
BC00226=212842,1022781,1075175
BC00227=146334,1015862,1075175
BC00228=66205,1045023,1075175
BC00229=66205,1045023,1075175
BC00230=66205,1045023,1075175
BC00231=66205,1045023,1075175
BC00232=66205,1045023,1075175
BC00233=66205,1045023,1075175
BC00234=66205,1045023,1075175
BC00235=66205,1045023,1075175
BC00236=66205,1045023,1075175
BC00237=66205,1045023,1075175
BC00238=66205,1045023,1075175
BC00239=66205,1045023,1075175
BC00240=125029,959783,1075175
BC00241=190390,972133,1075175
BC00242=190390,972133,1075175
BC00243=190390,972133,1075173
BC00244=190390,972133,1075175
BC00245=190390,972133,1075175
BC00246=190390,972133,1075175
BC00247=190390,972133,1075175
BC00248=190390,972133,1075175
BC00249=190390,972133,1075175
BC00250=190390,972133,1075175
BC00251=190390,972133,1075175
BC00252=190390,972133,1075175
BC00253=190390,972133,1075175
BC00254=103363,888035,1075175
BC00255=35304,822265,1075175
BC00256=35304,822265,1075175
BC00257=35304,822265,1075175
BC00258=35304,822265,1075175
BC00259=35304,822265,1075175
BC00260=35304,822265,1075175
BC00261=35304,822265,1075175
BC00262=35304,822265,1075175
BC00263=35304,822265,1075175
BC00264=35304,822265,1075175
BC00265=35304,822265,1075175
BC00266=35304,822265,1075175
BC00267=167967,799945,1075175
BC00268=311305,898961,1075175
BC00269=311305,898961,1075175
BC00270=311305,898961,1075175
BC00271=311305,898961,1075175
BC00272=311305,898961,1075175
BC00273=311305,898961,1075175
BC00274=311305,898961,1075175
BC00275=311305,898961,1075175
BC00276=311305,898961,1075175
BC00277=311305,898961,1075175
BC00278=311305,898961,1075175
BC00279=311305,898961,1075175
BC00280=113180,824290,1075229
BC00281=113180,824290,1075229
BC00282=113180,824290,1075229
BC00283=113180,824290,1075229
BC00284=113180,824290,1075229
BC00285=113180,824290,1075229
BC00286=113180,824290,1075229
BC00287=113180,824290,1075229
BC00288=113180,824290,1075229
BC00289=113180,824290,1075229
BC00290=113180,824290,1075229
BC00291=113180,824290,1075229
BC00292=355762,967535,1075175
BC00293=355762,967535,1075175
BC00294=355762,967535,1075175
BC00295=355762,967535,1075175
BC00296=355762,967535,1075175
BC00297=355762,967535,1075175
BC00298=355762,967535,1075175
BC00299=355762,967535,1075175
BC00300=397203,974799,1075175
BC00301=397203,974799,1075175
BC00302=397203,974799,1075175
BC00303=397203,974799,1075175
BC00304=397203,974799,1075175
BC00305=397203,974799,1075175
BC00306=397203,974799,1075175
BC00307=397203,974799,1075175
BC00308=279782,952911,1075175
BC00309=264332,967435,1075175
BC00310=264332,967435,1075175
BC00311=264332,967435,1075175
BC00312=264332,967435,1075175
BC00313=264332,967435,1075175
BC00314=264332,967435,1075175
BC00315=264332,967435,1075175
BC00316=264332,967435,1075175
BC00317=264332,967435,1075175
BC00318=264332,967435,1075175
BC00319=264332,967435,1075175
BC00320=290594,956201,1075175
BC00321=316856,944967,1075175
BC00322=316856,944967,1075175
BC00323=316856,944967,1075175
BC00324=316856,944967,1075175
BC00325=316856,944967,1075175
BC00326=316856,944967,1075175
BC00327=316856,944967,1075175
BC00328=316856,944967,1075175
BC00329=316856,944967,1075175
BC00330=316856,944967,1075175
BC00331=316856,944967,1075175
BC00332=316856,944967,1075175
BC00333=316856,944967,1075175
BC00334=316856,944967,1075175
BC00335=316856,944967,1075175
BC00336=316856,944967,1075175
BC00337=329946,891084,1075175
BC00338=337525,859888,1075175
BC00339=337525,859888,1075175
BC00340=337525,859888,1075175
BC00341=337525,859888,1075175
BC00342=337525,859888,1075175
BC00343=337525,859888,1075175
BC00344=337525,859888,1075175
BC00345=337525,859888,1075175
BC00346=238148,874377,1075175
BC00347=227206,875826,1075175
BC00348=227206,875826,1075175
BC00349=227206,875826,1075175
BC00350=227206,875826,1075175
BC00351=227206,875826,1075175
BC00352=227206,875826,1075175
BC00353=280946,887675,1075175
BC00354=280946,887675,1075175
BC00355=280946,887675,1075175
BC00356=280946,887675,1075175
BC00357=280946,887675,1075175
BC00358=280946,887675,1075175
BC00359=280946,887675,1075175
BC00360=280946,887675,1075175
BC00361=239261,850045,1075175
BC00362=207869,857354,1075175
BC00363=207869,857354,1075175
BC00364=207869,857354,1075175
BC00365=207869,857354,1075175
BC00366=207869,857354,1075175
BC00367=207869,857354,1075175
BC00368=207869,857354,1075175
BC00369=207869,857354,1075175
BC00370=207996,857850,1075175
BC00371=184532,936508,1075175
BC00372=203495,1021788,1075175
BC00373=203934,1024782,1075175
BC00374=204109,1022908,1075172
BC00375=204109,1022908,1075172
BC00376=193998,1019034,1075175
BC00377=193559,1023720,1075175
BC00378=122539,997675,1075175
BC00379=122539,997675,1075175
BC00380=122540,997675,1075169
BC00381=122540,997675,1075169
BC00382=122539,997675,1075175
BC00383=122539,997675,1075175
BC00384=110261,971952,1075175
BC00385=110261,971952,1075175
BC00386=110261,971952,1075175
BC00387=110261,971952,1075175
BC00388=110261,971952,1075175
BC00389=110261,971952,1075175
BC00390=222038,980891,1075175
BC00391=314817,1023461,1075175
BC00392=333143,1031869,1075175
BC00393=333143,1031869,1075175
BC00394=333143,1031869,1075175
BC00395=333143,1031869,1075175
BC00396=333143,1031869,1075175
BC00397=163675,1006427,1075175
BC00398=163675,1006427,1075175
BC00399=164114,1001741,1075175
BC00400=164289,999867,1075175
BC00401=160191,997498,1075175
BC00402=158450,996490,1075175
BC00403=154353,994119,1075175
BC00404=154178,995993,1075175
BC00405=153739,1000679,1075175
BC00406=82719,974634,1075175
BC00407=82719,974634,1075175
BC00408=82720,974634,1075172
BC00409=82720,974634,1075172
BC00410=82719,974634,1075175
BC00411=82720,974634,1075173
BC00412=82719,974634,1075175
BC00413=82719,974634,1075175
BC00414=70441,948911,1075175
BC00415=70441,948911,1075175
BC00416=70441,948911,1075175
BC00417=70441,948911,1075175
BC00418=70441,948911,1075175
BC00419=70441,948911,1075175
BC00420=182218,957850,1075175
BC00421=274997,1000420,1075175
BC00422=293323,1008828,1075175
BC00423=293323,1008828,1075175
BC00424=293323,1008828,1075175
BC00425=293323,1008828,1075175
BC00426=293323,1008828,1075175
BC00427=293323,1008828,1075175
BC00428=337244,1059629,1075175
BC00429=337244,1059629,1075175
BC00430=337244,1059629,1075175
BC00431=337244,1059629,1075175
BC00432=337244,1059629,1075175
BC00433=337244,1059629,1075175
BC00434=337244,1059629,1075175
BC00435=227430,982125,1075175
BC00436=115014,939685,1075175
BC00437=118867,937244,1075175
BC00438=120408,936268,1075175
BC00439=140995,947826,1075175
BC00440=182041,976368,1075175
BC00441=180846,977671,1075175
BC00442=177859,980929,1075175
BC00443=194800,984537,1075175
BC00444=244653,1016084,1075175
BC00445=241511,1010564,1075175
BC00446=240254,1008357,1075175
BC00447=240254,1008354,1075175
BC00448=241511,1010562,1075175
BC00449=244653,1016081,1075175
BC00450=244653,1016084,1075175
BC00451=272695,1033702,1075175
BC00452=285514,1041756,1075175
BC00453=284751,1045931,1075175
BC00454=282162,1039999,1075175
BC00455=281126,1037626,1075175
BC00456=207140,1028015,1075175
BC00457=213441,1031536,1075175
BC00458=213388,1030834,1075175
BC00459=213388,1030834,1075175
BC00460=212628,1031081,1075217
BC00461=212628,1031081,1075217
BC00462=212628,1031081,1075217
BC00463=212628,1031081,1075217
BC00464=212628,1031081,1075202
BC00465=202210,1012854,1075175
BC00466=202210,1012854,1075175
BC00467=196613,982513,1075175
BC00468=175963,870568,1075175
BC00469=163612,803610,1075175
BC00470=152631,778532,1075175
BC00471=146092,780306,1075175
BC00472=143477,781016,1075175
BC00473=143597,781078,1075175
BC00474=143625,781092,1075175
BC00475=143746,781156,1075175
BC00476=146361,780446,1075175
BC00477=152900,778672,1075175
BC00478=152900,778672,1075175
BC00479=74084,744686,1075175
BC00480=74084,744686,1075175
BC00481=67287,679894,1075175
BC00482=67287,679894,1075175
BC00483=67287,679894,1075175
BC00484=67287,679894,1075175
BC00485=67287,679894,1075175
BC00486=67287,679894,1075175
BC00487=67287,679894,1075175
BC00488=67287,679894,1075175
BC00489=83395,694294,1075175
BC00490=102108,711022,1075175
BC00491=165558,767742,1075175
BC00492=222482,818628,1075175
BC00493=215814,820321,1075175
BC00494=213147,820999,1075175
BC00495=213147,820994,1075175
BC00496=213147,820993,1075175
BC00497=213148,820988,1075175
BC00498=215815,820311,1075175
BC00499=222483,818617,1075175
BC00500=173722,816110,1075175
BC00501=90356,811823,1075175
BC00502=89696,811574,1075175
BC00503=89432,811475,1075175
BC00504=85301,809160,1075175
BC00505=73323,802435,1075175
BC00506=69196,800114,1075175
BC00507=69460,800213,1075175
BC00508=70120,800462,1075175
BC00509=203969,867991,1075175
BC00510=200192,866637,1075175
BC00511=198681,866095,1075175
BC00512=196278,870078,1075175
BC00513=188025,883752,1075175
BC00514=185620,887734,1075175
BC00515=187131,888276,1075175
BC00516=190907,889630,1075175
BC00517=185807,834457,1075175
BC00518=185042,826181,1075175
BC00519=182820,831186,1075175
BC00520=181931,833188,1075175
BC00521=205283,846231,1075175
BC00522=246906,863634,1075175
BC00523=246906,863634,1075175
BC00524=248214,861732,1075175
BC00525=251484,856977,1075175
BC00526=177002,833071,1075175
BC00527=153563,828435,1075175
BC00528=140020,825224,1075175
BC00529=143607,831260,1075175
BC00530=145042,833675,1075175
BC00531=145042,833669,1075175
BC00532=143607,831255,1075175
BC00533=140021,825218,1075175
BC00534=140020,825224,1075175
BC00535=325300,955877,1075175
BC00536=326098,960603,1075175
BC00537=326417,962494,1075175
BC00538=373942,970744,1075175
BC00539=373623,968854,1075175
BC00540=372825,964128,1075175
BC00541=388713,844195,1075175
BC00542=388713,844195,1075175
BC00543=388713,844195,1075175
BC00544=388713,844195,1075175
BC00545=388713,844195,1075175
BC00546=392621,845560,1075175
BC00547=388844,869736,1075175
BC00548=388844,869736,1075175
BC00549=388844,869736,1075175
BC00550=388844,869736,1075175
BC00551=386515,859937,1075175
BC00552=382579,861240,1075175
BC00553=382579,861240,1075175
BC00554=398174,862085,1075175
BC00555=398174,860729,1075175
BC00556=398175,860364,1075172
BC00557=398174,860364,1075175
BC00558=398174,860364,1075175
BC00559=398174,860364,1075175
BC00560=398174,859798,1075175
BC00561=398174,853900,1075175
BC00562=335556,962122,1075175
BC00563=313093,960913,1075175
BC00564=312779,966350,1075175
BC00565=312653,968525,1075175
BC00566=317356,969341,1075175
BC00567=322596,970251,1075175
BC00568=322722,968076,1075175
BC00569=323035,962639,1075175
BC00570=275790,965253,1075175
BC00571=219096,968390,1075175
BC00572=223120,970377,1075175
BC00573=224729,971172,1075175
BC00574=220819,966503,1075175
BC00575=219210,965708,1075175
BC00576=215186,963721,1075175
BC00577=283252,975030,1075175
BC00578=343583,985054,1075175
BC00579=351318,986339,1075175
BC00580=346951,987672,1075175
BC00581=345577,987893,1075175
BC00582=346840,986833,1075175
BC00583=348087,985787,1075175
BC00584=349722,984415,1075175
BC00585=349722,984415,1075175
BC00586=349722,984415,1075175
BC00587=351469,983882,1075175
BC00588=355836,982549,1075175
BC00589=351318,986339,1075175
BC00590=375376,962122,1075175
BC00591=352913,960913,1075175
BC00592=352599,966350,1075175
BC00593=352473,968525,1075175
BC00594=357176,969341,1075175
BC00595=362416,970251,1075175
BC00596=362542,968076,1075175
BC00597=362855,962639,1075175
BC00598=315610,965253,1075175
BC00599=258916,968390,1075175
BC00600=262940,970377,1075175
BC00601=264549,971172,1075175
BC00602=260639,966503,1075175
BC00603=259030,965708,1075175
BC00604=255006,963721,1075175
BC00605=323072,975030,1075175
BC00606=383403,985054,1075175
BC00607=391138,986339,1075175
BC00608=386771,987672,1075175
BC00609=385397,987893,1075175
BC00610=386660,986833,1075175
BC00611=387907,985787,1075175
BC00612=389542,984415,1075175
BC00613=389542,984415,1075175
BC00614=389542,984415,1075175
BC00615=391289,983882,1075175
BC00616=394785,983280,1075175
BC00617=393350,984484,1075175
BC00618=322594,894090,1075175
BC00619=319270,885244,1075175
BC00620=319145,881395,1075175
BC00621=319096,879856,1075175
BC00622=319096,879856,1075175
BC00623=310158,881364,1075175
BC00624=310282,885213,1075175
BC00625=287932,898047,1075175
BC00626=289217,893542,1075175
BC00627=289730,891739,1075175
BC00628=285692,891718,1075175
BC00629=285179,893520,1075175
BC00630=283894,898026,1075175
BC00631=317886,904348,1075175
BC00632=321408,904356,1075175
BC00633=251917,914686,1075175
BC00634=191223,885215,1075175
BC00635=191223,923708,1075175
BC00636=186619,926680,1075175
BC00637=184777,927869,1075175
BC00638=132357,904545,1075175
BC00639=148459,907340,1075175
BC00640=150318,907039,1075175
BC00641=172119,903510,1075175
BC00642=172334,901853,1075175
BC00643=172871,897709,1075175
BC00644=285135,920733,1075175
BC00645=282294,924718,1075175
BC00646=278369,925274,1075175
BC00647=250842,915028,1075175
BC00648=259644,916574,1075175
BC00649=259644,916574,1075175
BC00650=259644,916574,1075175
BC00651=285135,920733,1075175
BC00652=320470,920733,1075175
BC00653=320470,920733,1075175
BC00654=320470,920733,1075172
BC00655=320470,920733,1075172
BC00656=320470,920733,1075172
BC00657=302481,924098,1075175
BC00658=235391,926007,1075175
BC00659=235391,926007,1075175
BC00660=227742,920504,1075175
BC00661=172871,874776,1075175
BC00662=140749,823212,1075175
BC00663=114392,780903,1075175
BC00664=114392,780903,1075175
BC00665=114392,780903,1075175
BC00666=114392,780903,1075175
BC00667=114392,780903,1075175
BC00668=114392,780903,1075175
BC00669=114392,780903,1075175
BC00670=114392,780903,1075175
BC00671=147421,791636,1075175
BC00672=157474,794903,1075175
BC00673=157474,794903,1075175
BC00674=157474,794903,1075175
BC00675=157474,794903,1075175
BC00676=157474,794903,1075175
BC00677=157474,794903,1075175
BC00678=157474,794903,1075175
BC00679=157474,794903,1075175
BC00680=188976,808930,1075175
BC00681=188976,808930,1075175
BC00682=188976,808930,1075175
BC00683=188976,808930,1075175
BC00684=188976,808930,1075175
BC00685=188976,808930,1075175
BC00686=188976,808930,1075175
BC00687=188976,808930,1075175
BC00688=147641,782026,1075175
BC00689=198576,845167,1075175
BC00690=232811,933878,1075175
BC00691=232896,933343,1075175
BC00692=232035,938717,1075175
BC00693=231691,940867,1075175
BC00694=233684,941999,1075172
BC00695=218918,951560,1075175
BC00696=218487,945823,1075175
BC00697=199715,965567,1075175
BC00698=202231,971242,1075175
BC00699=203237,973512,1075175
BC00700=199770,971953,1075175
BC00701=198686,969649,1075175
BC00702=195975,963887,1075175
BC00703=268319,958805,1075175
BC00704=299772,956595,1075175
BC00705=294961,960779,1075175
BC00706=302025,967105,1075175
BC00707=302025,967105,1075175
BC00708=302862,967571,1075175
BC00709=304981,965989,1075175
BC00710=310277,962032,1075175
BC00711=299772,946803,1075175
BC00712=156368,867370,1075175
BC00713=114190,943890,1075175
BC00714=112857,947238,1075175
BC00715=112324,948578,1075175
BC00716=57438,939049,1075175
BC00717=57438,939049,1075175
BC00718=57972,937710,1075175
BC00719=59304,934362,1075175
BC00720=59959,931573,1075175
BC00721=60163,930702,1075175
BC00722=64900,934429,1075175
BC00723=66794,935919,1075175
BC00724=70926,933782,1075175
BC00725=86714,920781,1075175
BC00726=88876,916896,1075175
BC00727=87247,915034,1075175
BC00728=83174,910378,1075175
BC00729=93083,910762,1075175
BC00730=96362,916987,1075175
BC00731=97673,919477,1075175
BC00732=102107,915596,1075175
BC00733=93734,925368,1075175
BC00734=92128,923198,1075175
BC00735=88115,917772,1075175
BC00736=59304,853852,1075175
BC00737=302197,956351,1075175
BC00738=302197,956351,1075175
BC00739=297684,958955,1075175
BC00740=295879,959997,1075175
BC00741=304739,998959,1075175
BC00742=304723,978619,1075175
BC00743=293949,1042099,1075175
BC00744=295296,1044279,1075175
BC00745=298665,1049727,1075175
BC00746=298665,1049727,1075175
BC00747=302197,956351,1075175
BC00748=339931,956351,1075175
BC00749=339931,956351,1075175
BC00750=339931,956351,1075175
BC00751=345108,996833,1075175
BC00752=329498,1037164,1075167
BC00753=329498,1037164,1075167
BC00754=326051,1024211,1075168
BC00755=315665,949153,1075168
BC00756=252444,896504,1075168
BC00757=116643,896504,1075168
BC00758=116643,972299,1075168
BC00759=116644,972299,1070754
BC00760=116644,972299,1070754
BC00761=121804,1001122,1070754
BC00762=121804,1001122,1070754
BC00763=121804,1001122,1070754
BC00764=121804,1001122,1070754
BC00765=164206,909682,1070754
BC00766=118737,834368,1072160
BC00767=21214,672831,1075175
BC00768=21214,672831,272422
BC00769=236199,677421,175874
BC00770=277013,737492,108841
BC00771=313151,790681,49489
BC00772=313151,790681,49489
BC00773=313151,790681,49489
BC00774=313151,790681,49489
BC00775=313151,790681,49489
BC00776=313151,790681,49489
BC00777=313151,790681,49489
BC00778=313151,790681,49489
BC00779=313151,790681,49489
BC00780=339082,790681,219047
BC00781=339082,790681,219047
BC00782=339082,790681,219047
BC00783=339082,790681,219047
BC00784=339082,790681,219047
BC00785=339082,790681,219047
BC00786=339082,790681,219047
BC00787=339082,790681,219047
BC00788=339082,790681,219047
BC00789=318756,790681,206942
BC00790=318756,790681,206942
BC00791=318756,790681,206942
BC00792=318756,790681,206942
BC00793=318756,790681,206942
BC00794=318756,790681,206942
BC00795=318756,790681,206941
BC00796=318756,790681,206941
BC00797=318756,790681,206942
BC00798=330178,790681,186109
BC00799=360333,790681,131110
BC00800=360333,790681,131110
BC00801=360333,790681,131110
BC00802=360333,790681,131110
BC00803=360333,790681,131110
BC00804=360333,790681,131110
BC00805=360333,790681,131110
BC00806=360333,790681,131110
BC00807=360333,790681,131110
BC00808=319787,790681,204440
BC00809=319787,790681,204440
BC00810=319787,790681,204440
BC00811=319787,790681,204440
BC00812=319787,790681,204440
BC00813=319787,790681,204440
BC00814=319787,790681,204440
BC00815=319787,790681,204440
BC00816=319787,790681,204440
BC00817=319787,790681,204440
BC00818=345989,790681,139065
BC00819=345989,790681,139065
BC00820=345989,790681,139065
BC00821=345989,790681,139065
BC00822=345989,790681,139065
BC00823=345989,790681,139065
BC00824=345989,790681,139065
BC00825=345989,790681,139065
BC00826=345989,790681,139065
BC00827=308625,748445,196549
BC00828=237635,668196,305769
BC00829=196160,672502,403752
BC00830=196160,672502,403752
BC00831=196160,727236,321537
BC00832=196160,765129,264619
BC00833=196160,765129,264619
BC00834=196160,765129,264619
BC00835=196160,765129,264619
BC00836=196160,765129,264619
BC00837=196160,765129,264619
BC00838=196160,765129,264619
BC00839=196160,765129,264619
BC00840=196160,765129,264619
BC00841=196160,765129,264619
BC00842=172117,778418,210988
BC00843=172117,778418,210988
BC00844=172117,778418,210988
BC00845=172117,778418,210988
BC00846=172117,778418,210988
BC00847=172117,778418,210988
BC00848=172117,778418,210988
BC00849=172117,778418,210988
BC00850=172117,778418,210988
BC00851=149065,790681,133702
BC00852=149065,790681,133702
BC00853=149065,790681,133702
BC00854=149065,790681,133702
BC00855=149065,790681,133702
BC00856=149065,790681,133702
BC00857=149065,790681,133702
BC00858=149065,790681,133702
BC00859=149065,790681,133702
BC00860=149065,790681,133702
BC00861=149065,790681,133702
BC00862=149065,790681,133702
BC00863=117513,790681,53
BC00864=117513,790681,53
BC00865=117513,790681,53
BC00866=117513,790681,53
BC00867=117513,790681,53
BC00868=117513,790681,53
BC00869=117513,790681,53
BC00870=117513,790681,53
BC00871=117513,790681,53
BC00872=117513,790681,53
BC00873=117513,790681,53
BC00874=117513,790681,53
BC00875=117513,790681,53
BC00876=190612,790681,158488
BC00877=190612,790681,158488
BC00878=190612,790681,158488
BC00879=190612,790681,158488
BC00880=190612,790681,158488
BC00881=190612,790681,158488
BC00882=184906,790681,111068
BC00883=184906,790681,111068
BC00884=184906,790681,111068
BC00885=184906,790681,111068
BC00886=184906,790681,111068
BC00887=184906,790681,111068
BC00888=181347,790681,153019
BC00889=174520,790681,233505
BC00890=174520,790681,233505
BC00891=174520,790681,233505
BC00892=174520,790681,233505
BC00893=174520,790681,233505
BC00894=174520,790681,233505
BC00895=184991,733498,315883
BC00896=196160,672502,403752
BC00897=196160,672502,403752
BC00898=237635,668196,305769
BC00899=308625,748445,196549
BC00900=309549,790681,184299
BC00901=309549,790681,184299
BC00902=309549,790681,184299
BC00903=309549,790681,184299
BC00904=309549,790681,184299
BC00905=309549,790681,184299
BC00906=321199,790681,207159
BC00907=321199,790681,207159
BC00908=321199,790681,207159
BC00909=321199,790681,207159
BC00910=321199,790681,207159
BC00911=321199,790681,207159
BC00912=321199,790681,207159
BC00913=321199,790681,207159
BC00914=373020,790681,107875
BC00915=373020,790681,107875
BC00916=373020,790681,107875
BC00917=373020,790681,107875
BC00918=373020,790681,107875
BC00919=373020,790681,107875
BC00920=373020,790681,107875
BC00921=373020,790681,107875
BC00922=367447,763418,217217
BC00923=362764,784495,185132
BC00924=361390,790681,53
BC00925=361390,790681,53
BC00926=361390,790681,53
BC00927=361390,790681,53
BC00928=361390,790681,53
BC00929=361390,790681,53
BC00930=340769,790681,53
BC00931=340769,790681,53
BC00932=340769,790681,53
BC00933=340769,790681,53
BC00934=340769,790681,53
BC00935=340769,790681,53
BC00936=340769,790681,53
BC00937=340769,790681,53
BC00938=340769,790681,53
BC00939=340769,790681,53
BC00940=340769,790681,53
BC00941=340769,790681,53
BC00942=340769,790681,53
BC00943=340769,790681,53
BC00944=340769,790681,53
BC00945=340769,765105,53
BC00946=340769,765105,53
BC00947=340769,765105,53
BC00948=340769,765105,53
BC00949=340769,765105,53
BC00950=340769,765105,53
BC00951=340769,765105,53
BC00952=326290,746662,147117
BC00953=300313,667687,410966
BC00954=300313,667687,410966
BC00955=200178,761203,279737
BC00956=168613,790681,238372
BC00957=168613,790681,238372
BC00958=168613,790681,238372
BC00959=168613,790681,238372
BC00960=168613,790681,238372
BC00961=168613,790681,238372
BC00962=187396,785580,192031
BC00963=187396,785580,192031
BC00964=187396,785580,192031
BC00965=187396,785580,192031
BC00966=187396,785580,192031
BC00967=187396,785580,192031
BC00968=200178,761203,279737
BC00969=300313,667687,410966
BC00970=300313,667687,410966
BC00971=326290,746662,147117
BC00972=326023,790681,196549
BC00973=326023,790681,196549
BC00974=326023,790681,196549
BC00975=326023,790681,196549
BC00976=326023,790681,196549
BC00977=326023,790681,196549
BC00978=316509,790681,152288
BC00979=316509,790681,152288
BC00980=316509,790681,152288
BC00981=316509,790681,152288
BC00982=316509,790681,152288
BC00983=316509,790681,152288
BC00984=314401,774670,185962
BC00985=300313,667687,410966
BC00986=300313,667687,410966
BC00987=200178,761203,279737
BC00988=186958,779092,256601
BC00989=178395,790681,241614
BC00990=178395,790681,241614
BC00991=178395,790681,241614
BC00992=178395,790681,241614
BC00993=178395,790681,241614
BC00994=178395,790681,241614
BC00995=198041,770354,161044
BC00996=198041,770354,161044
BC00997=198041,770354,161044
BC00998=198041,770354,161044
BC00999=198041,770354,161044
BC01000=198041,770354,161044
BC01001=200178,761203,279737
BC01002=300313,667687,410966
BC01003=300313,667687,410966
BC01004=363254,767093,179444
BC01005=378190,790681,124507
BC01006=378190,790681,124507
BC01007=378190,790681,124507
BC01008=378190,790681,124507
BC01009=378190,790681,124507
BC01010=378190,790681,124507
BC01011=345239,790681,222063
BC01012=345239,790681,222063
BC01013=345239,790681,222063
BC01014=345239,790681,222063
BC01015=345239,790681,222063
BC01016=345239,790681,222063
BC01017=363254,767093,179444
BC01018=300313,667687,410966
BC01019=300313,667687,410966
BC01020=200178,761203,279737
BC01021=142668,790681,138813
BC01022=142668,790681,138813
BC01023=142668,790681,138813
BC01024=142668,790681,138813
BC01025=142668,790681,138813
BC01026=142668,790681,138813
BC01027=142668,790681,138813
BC01028=142668,790681,138813
BC01029=203164,773756,23252
BC01030=203164,773756,23252
BC01031=203164,773756,23252
BC01032=203164,773756,23252
BC01033=203164,773756,23252
BC01034=203164,773756,23252
BC01035=200599,780936,88057
BC01036=197119,790681,176008
BC01037=197119,790681,176008
BC01038=197119,790681,176008
BC01039=197119,790681,176008
BC01040=197119,790681,176008
BC01041=197119,790681,176008
BC01042=197993,782258,205645
BC01043=199960,763308,272330
BC01044=201592,760202,280395
BC01045=200178,669563,279737
BC01046=78393,670967,1075175
EC00000=798156,0
EC00001=798153,3
EC00002=798156,0
EC00003=798156,0
EC00004=798156,0
EC00005=798156,0
EC00006=798156,0
EC00007=798156,0
EC00008=798156,0
EC00009=798156,0
EC00010=798156,0
EC00011=798156,0
EC00012=798156,0
EC00013=798156,0
EC00014=798156,0
EC00015=798156,0
EC00016=798156,0
EC00017=798156,0
EC00018=798156,0
EC00019=798156,0
EC00020=798156,0
EC00021=798156,0
EC00022=798156,0
EC00023=798156,0
EC00024=798156,0
EC00025=798156,0
EC00026=798156,0
EC00027=798156,0
EC00028=798156,0
EC00029=798156,0
EC00030=798156,0
EC00031=798156,0
EC00032=798156,0
EC00033=798156,0
EC00034=798156,0
EC00035=798156,0
EC00036=798156,0
EC00037=798156,0
EC00038=798156,0
EC00039=798156,0
EC00040=798156,0
EC00041=798156,0
EC00042=798156,0
EC00043=798156,0
EC00044=798156,0
EC00045=798156,0
EC00046=798156,0
EC00047=798156,0
EC00048=798156,0
EC00049=798156,0
EC00050=798156,0
EC00051=798156,0
EC00052=798156,0
EC00053=798156,0
EC00054=798156,0
EC00055=798156,0
EC00056=798156,0
EC00057=798156,0
EC00058=798156,0
EC00059=798156,0
EC00060=798156,0
EC00061=798156,0
EC00062=798156,0
EC00063=798156,0
EC00064=798156,0
EC00065=798156,0
EC00066=798156,0
EC00067=798156,0
EC00068=798156,0
EC00069=798156,0
EC00070=798156,0
EC00071=798156,0
EC00072=798156,0
EC00073=798156,0
EC00074=798156,0
EC00075=798156,0
EC00076=798156,0
EC00077=798156,0
EC00078=798156,0
EC00079=798156,0
EC00080=798156,0
EC00081=798156,0
EC00082=798156,0
EC00083=798156,0
EC00084=798156,0
EC00085=798156,0
EC00086=798156,0
EC00087=798156,0
EC00088=798156,0
EC00089=798156,0
EC00090=798156,0
EC00091=798156,0
EC00092=798156,0
EC00093=798156,0
EC00094=798156,0
EC00095=798156,0
EC00096=798156,0
EC00097=798156,0
EC00098=798156,0
EC00099=798156,0
EC00100=798156,0
EC00101=798156,0
EC00102=798156,0
EC00103=798156,0
EC00104=798156,0
EC00105=798156,0
EC00106=798156,0
EC00107=798156,0
EC00108=798156,0
EC00109=798156,0
EC00110=798156,0
EC00111=798156,0
EC00112=798156,0
EC00113=798156,0
EC00114=798156,0
EC00115=798155,0
EC00116=798155,0
EC00117=798155,0
EC00118=798155,0
EC00119=798155,0
EC00120=798155,0
EC00121=798155,0
EC00122=798155,0
EC00123=798155,0
EC00124=798156,0
EC00125=798156,0
EC00126=798156,0
EC00127=798156,0
EC00128=798156,0
EC00129=798156,0
EC00130=798156,0
EC00131=798156,0
EC00132=798156,0
EC00133=798156,0
EC00134=798156,0
EC00135=798156,0
EC00136=798156,0
EC00137=798156,0
EC00138=798156,0
EC00139=798156,0
EC00140=798156,0
EC00141=798156,0
EC00142=798156,0
EC00143=798156,0
EC00144=798156,0
EC00145=798156,0
EC00146=798156,0
EC00147=798156,0
EC00148=798156,0
EC00149=798156,0
EC00150=798156,0
EC00151=798156,0
EC00152=798156,0
EC00153=798156,0
EC00154=798156,0
EC00155=798156,0
EC00156=798156,0
EC00157=798156,0
EC00158=798156,0
EC00159=798156,0
EC00160=798156,0
EC00161=798156,0
EC00162=798156,0
EC00163=798156,0
EC00164=798156,0
EC00165=798156,0
EC00166=798156,0
EC00167=798156,0
EC00168=798156,0
EC00169=798156,0
EC00170=798156,0
EC00171=798156,0
EC00172=798156,0
EC00173=798156,0
EC00174=798156,0
EC00175=798156,0
EC00176=798156,0
EC00177=798156,0
EC00178=798156,0
EC00179=798156,0
EC00180=798156,0
EC00181=798156,0
EC00182=798156,0
EC00183=798156,0
EC00184=798156,0
EC00185=798156,0
EC00186=798156,0
EC00187=798156,0
EC00188=798156,0
EC00189=798156,0
EC00190=798156,0
EC00191=798156,0
EC00192=798156,0
EC00193=798156,0
EC00194=798156,0
EC00195=798156,0
EC00196=798156,0
EC00197=798156,0
EC00198=798156,0
EC00199=798156,0
EC00200=798156,0
EC00201=798156,0
EC00202=798156,0
EC00203=798156,0
EC00204=798156,0
EC00205=798156,0
EC00206=798156,0
EC00207=798156,0
EC00208=798156,0
EC00209=798156,0
EC00210=798156,0
EC00211=798156,0
EC00212=798156,0
EC00213=798156,0
EC00214=798156,0
EC00215=798156,0
EC00216=798156,0
EC00217=798156,0
EC00218=798156,0
EC00219=798156,0
EC00220=798156,0
EC00221=798156,0
EC00222=798156,0
EC00223=798156,0
EC00224=798156,0
EC00225=798156,0
EC00226=798156,0
EC00227=798156,0
EC00228=798156,0
EC00229=798156,0
EC00230=798156,0
EC00231=798156,0
EC00232=798156,0
EC00233=798156,0
EC00234=798156,0
EC00235=798156,0
EC00236=798156,0
EC00237=798156,0
EC00238=798156,0
EC00239=798156,0
EC00240=798156,0
EC00241=798156,0
EC00242=798156,0
EC00243=798154,2
EC00244=798156,0
EC00245=798156,0
EC00246=798156,0
EC00247=798156,0
EC00248=798156,0
EC00249=798156,0
EC00250=798156,0
EC00251=798156,0
EC00252=798156,0
EC00253=798156,0
EC00254=798156,0
EC00255=798156,0
EC00256=798156,0
EC00257=798156,0
EC00258=798156,0
EC00259=798156,0
EC00260=798156,0
EC00261=798156,0
EC00262=798156,0
EC00263=798156,0
EC00264=798156,0
EC00265=798156,0
EC00266=798156,0
EC00267=798156,0
EC00268=798156,0
EC00269=798156,0
EC00270=798156,0
EC00271=798156,0
EC00272=798156,0
EC00273=798156,0
EC00274=798156,0
EC00275=798156,0
EC00276=798156,0
EC00277=798156,0
EC00278=798156,0
EC00279=798156,0
EC00280=798156,0
EC00281=798156,0
EC00282=798156,0
EC00283=798156,0
EC00284=798156,0
EC00285=798156,0
EC00286=798156,0
EC00287=798156,0
EC00288=798156,0
EC00289=798156,0
EC00290=798156,0
EC00291=798156,0
EC00292=798156,0
EC00293=798156,0
EC00294=798156,0
EC00295=798156,0
EC00296=798156,0
EC00297=798156,0
EC00298=798156,0
EC00299=798156,0
EC00300=798156,0
EC00301=798156,0
EC00302=798156,0
EC00303=798156,0
EC00304=798156,0
EC00305=798156,0
EC00306=798156,0
EC00307=798156,0
EC00308=798156,0
EC00309=798156,0
EC00310=798156,0
EC00311=798156,0
EC00312=798156,0
EC00313=798156,0
EC00314=798156,0
EC00315=798156,0
EC00316=798156,0
EC00317=798156,0
EC00318=798156,0
EC00319=798156,0
EC00320=798156,0
EC00321=798156,0
EC00322=798156,0
EC00323=798156,0
EC00324=798156,0
EC00325=798156,0
EC00326=798156,0
EC00327=798156,0
EC00328=798156,0
EC00329=798156,0
EC00330=798156,0
EC00331=798156,0
EC00332=798156,0
EC00333=798156,0
EC00334=798156,0
EC00335=798156,0
EC00336=798156,0
EC00337=798156,0
EC00338=798156,0
EC00339=798156,0
EC00340=798156,0
EC00341=798156,0
EC00342=798156,0
EC00343=798156,0
EC00344=798156,0
EC00345=798156,0
EC00346=798156,0
EC00347=798156,0
EC00348=798156,0
EC00349=798156,0
EC00350=798156,0
EC00351=798156,0
EC00352=798156,0
EC00353=798156,0
EC00354=798156,0
EC00355=798156,0
EC00356=798156,0
EC00357=798156,0
EC00358=798156,0
EC00359=798156,0
EC00360=798156,0
EC00361=798156,0
EC00362=798156,0
EC00363=798156,0
EC00364=798156,0
EC00365=798156,0
EC00366=798156,0
EC00367=798156,0
EC00368=798156,0
EC00369=798156,0
EC00370=798156,0
EC00371=798156,0
EC00372=798156,0
EC00373=798156,0
EC00374=798155,0
EC00375=798155,0
EC00376=798156,0
EC00377=798156,0
EC00378=798156,0
EC00379=798156,0
EC00380=798154,0
EC00381=798154,0
EC00382=798156,0
EC00383=798156,0
EC00384=798156,0
EC00385=798156,0
EC00386=798156,0
EC00387=798156,0
EC00388=798156,0
EC00389=798156,0
EC00390=798156,0
EC00391=798156,0
EC00392=798156,0
EC00393=798156,0
EC00394=798156,0
EC00395=798156,0
EC00396=798156,0
EC00397=798156,0
EC00398=798156,0
EC00399=798156,0
EC00400=798156,0
EC00401=798156,0
EC00402=798156,0
EC00403=798156,0
EC00404=798156,0
EC00405=798156,0
EC00406=798156,0
EC00407=798156,0
EC00408=798155,0
EC00409=798155,0
EC00410=798156,0
EC00411=798155,0
EC00412=798156,0
EC00413=798156,0
EC00414=798156,0
EC00415=798156,0
EC00416=798156,0
EC00417=798156,0
EC00418=798156,0
EC00419=798156,0
EC00420=798156,0
EC00421=798156,0
EC00422=798156,0
EC00423=798156,0
EC00424=798156,0
EC00425=798156,0
EC00426=798156,0
EC00427=798156,0
EC00428=798156,0
EC00429=798156,0
EC00430=798156,0
EC00431=798156,0
EC00432=798156,0
EC00433=798156,0
EC00434=798156,0
EC00435=798156,0
EC00436=798156,0
EC00437=798156,0
EC00438=798156,0
EC00439=798156,0
EC00440=798156,0
EC00441=798156,0
EC00442=798156,0
EC00443=798156,0
EC00444=798156,0
EC00445=798156,0
EC00446=798156,0
EC00447=798156,0
EC00448=798156,0
EC00449=798156,0
EC00450=798156,0
EC00451=798156,0
EC00452=798156,0
EC00453=798156,0
EC00454=798156,0
EC00455=798156,0
EC00456=798156,0
EC00457=798156,0
EC00458=798156,0
EC00459=798156,0
EC00460=798154,1
EC00461=798154,1
EC00462=798154,1
EC00463=798154,1
EC00464=798151,2
EC00465=798156,0
EC00466=798156,0
EC00467=798156,0
EC00468=798156,0
EC00469=798156,0
EC00470=798156,0
EC00471=798156,0
EC00472=798156,0
EC00473=798156,0
EC00474=798156,0
EC00475=798156,0
EC00476=798156,0
EC00477=798156,0
EC00478=798156,0
EC00479=798156,0
EC00480=798156,0
EC00481=798156,0
EC00482=798156,0
EC00483=798156,0
EC00484=798156,0
EC00485=798156,0
EC00486=798156,0
EC00487=798156,0
EC00488=798156,0
EC00489=798156,0
EC00490=798156,0
EC00491=798156,0
EC00492=798156,0
EC00493=798156,0
EC00494=798156,0
EC00495=798156,0
EC00496=798156,0
EC00497=798156,0
EC00498=798156,0
EC00499=798156,0
EC00500=798156,0
EC00501=798156,0
EC00502=798156,0
EC00503=798156,0
EC00504=798156,0
EC00505=798156,0
EC00506=798156,0
EC00507=798156,0
EC00508=798156,0
EC00509=798156,0
EC00510=798156,0
EC00511=798156,0
EC00512=798156,0
EC00513=798156,0
EC00514=798156,0
EC00515=798156,0
EC00516=798156,0
EC00517=798156,0
EC00518=798156,0
EC00519=798156,0
EC00520=798156,0
EC00521=798156,0
EC00522=798156,0
EC00523=798156,0
EC00524=798156,0
EC00525=798156,0
EC00526=798156,0
EC00527=798156,0
EC00528=798156,0
EC00529=798156,0
EC00530=798156,0
EC00531=798156,0
EC00532=798156,0
EC00533=798156,0
EC00534=798156,0
EC00535=798156,0
EC00536=798156,0
EC00537=798156,0
EC00538=798156,0
EC00539=798156,0
EC00540=798156,0
EC00541=798156,0
EC00542=798156,0
EC00543=798156,0
EC00544=798156,0
EC00545=798156,0
EC00546=798156,0
EC00547=798156,0
EC00548=798156,0
EC00549=798156,0
EC00550=798156,0
EC00551=798156,0
EC00552=798156,0
EC00553=798156,0
EC00554=798156,0
EC00555=798156,0
EC00556=798156,1
EC00557=798156,0
EC00558=798156,0
EC00559=798156,0
EC00560=798156,0
EC00561=798156,0
EC00562=798156,0
EC00563=798156,0
EC00564=798156,0
EC00565=798156,0
EC00566=798156,0
EC00567=798156,0
EC00568=798156,0
EC00569=798156,0
EC00570=798156,0
EC00571=798156,0
EC00572=798156,0
EC00573=798156,0
EC00574=798156,0
EC00575=798156,0
EC00576=798156,0
EC00577=798156,0
EC00578=798156,0
EC00579=798156,0
EC00580=798156,0
EC00581=798156,0
EC00582=798156,0
EC00583=798156,0
EC00584=798156,0
EC00585=798156,0
EC00586=798156,0
EC00587=798156,0
EC00588=798156,0
EC00589=798156,0
EC00590=798156,0
EC00591=798156,0
EC00592=798156,0
EC00593=798156,0
EC00594=798156,0
EC00595=798156,0
EC00596=798156,0
EC00597=798156,0
EC00598=798156,0
EC00599=798156,0
EC00600=798156,0
EC00601=798156,0
EC00602=798156,0
EC00603=798156,0
EC00604=798156,0
EC00605=798156,0
EC00606=798156,0
EC00607=798156,0
EC00608=798156,0
EC00609=798156,0
EC00610=798156,0
EC00611=798156,0
EC00612=798156,0
EC00613=798156,0
EC00614=798156,0
EC00615=798156,0
EC00616=798156,0
EC00617=798156,0
EC00618=798156,0
EC00619=798156,0
EC00620=798156,0
EC00621=798156,0
EC00622=798156,0
EC00623=798156,0
EC00624=798156,0
EC00625=798156,0
EC00626=798156,0
EC00627=798156,0
EC00628=798156,0
EC00629=798156,0
EC00630=798156,0
EC00631=798156,0
EC00632=798156,0
EC00633=798156,0
EC00634=798156,0
EC00635=798156,0
EC00636=798156,0
EC00637=798156,0
EC00638=798156,0
EC00639=798156,0
EC00640=798156,0
EC00641=798156,0
EC00642=798156,0
EC00643=798156,0
EC00644=798156,0
EC00645=798156,0
EC00646=798156,0
EC00647=798156,0
EC00648=798156,0
EC00649=798156,0
EC00650=798156,0
EC00651=798156,0
EC00652=798156,0
EC00653=798156,0
EC00654=798155,1
EC00655=798155,1
EC00656=798155,1
EC00657=798156,0
EC00658=798156,0
EC00659=798156,0
EC00660=798156,0
EC00661=798156,0
EC00662=798156,0
EC00663=798156,0
EC00664=798156,0
EC00665=798156,0
EC00666=798156,0
EC00667=798156,0
EC00668=798156,0
EC00669=798156,0
EC00670=798156,0
EC00671=798156,0
EC00672=798156,0
EC00673=798156,0
EC00674=798156,0
EC00675=798156,0
EC00676=798156,0
EC00677=798156,0
EC00678=798156,0
EC00679=798156,0
EC00680=798156,0
EC00681=798156,0
EC00682=798156,0
EC00683=798156,0
EC00684=798156,0
EC00685=798156,0
EC00686=798156,0
EC00687=798156,0
EC00688=798156,0
EC00689=798156,0
EC00690=798156,0
EC00691=798156,0
EC00692=798156,0
EC00693=798156,0
EC00694=798155,0
EC00695=798156,0
EC00696=798156,0
EC00697=798156,0
EC00698=798156,0
EC00699=798156,0
EC00700=798156,0
EC00701=798156,0
EC00702=798156,0
EC00703=798156,0
EC00704=798156,0
EC00705=798156,0
EC00706=798156,0
EC00707=798156,0
EC00708=798156,0
EC00709=798156,0
EC00710=798156,0
EC00711=798156,0
EC00712=798156,0
EC00713=798156,0
EC00714=798156,0
EC00715=798156,0
EC00716=798156,0
EC00717=798156,0
EC00718=798156,0
EC00719=798156,0
EC00720=798156,0
EC00721=798156,0
EC00722=798156,0
EC00723=798156,0
EC00724=798156,0
EC00725=798156,0
EC00726=798156,0
EC00727=798156,0
EC00728=798156,0
EC00729=798156,0
EC00730=798156,0
EC00731=798156,0
EC00732=798156,0
EC00733=798156,0
EC00734=798156,0
EC00735=798156,0
EC00736=798156,0
EC00737=798156,0
EC00738=798156,0
EC00739=798156,0
EC00740=798156,0
EC00741=798156,0
EC00742=798156,0
EC00743=798156,0
EC00744=798156,0
EC00745=798156,0
EC00746=798156,0
EC00747=798156,0
EC00748=798156,0
EC00749=798156,0
EC00750=798156,0
EC00751=798156,0
EC00752=798153,2
EC00753=798153,2
EC00754=798153,2
EC00755=798153,2
EC00756=798153,2
EC00757=798153,2
EC00758=798153,2
EC00759=798152,2
EC00760=798152,2
EC00761=798152,2
EC00762=798152,2
EC00763=798152,2
EC00764=798152,2
EC00765=798152,2
EC00766=798153,1
EC00767=798156,0
EC00768=798156,0
EC00769=798156,0
EC00770=798156,0
EC00771=798156,0
EC00772=798156,0
EC00773=798156,0
EC00774=798156,0
EC00775=798156,0
EC00776=798156,0
EC00777=798156,0
EC00778=798156,0
EC00779=798156,0
EC00780=798156,0
EC00781=798156,0
EC00782=798156,0
EC00783=798156,0
EC00784=798156,0
EC00785=798156,0
EC00786=798156,0
EC00787=798156,0
EC00788=798156,0
EC00789=798156,0
EC00790=798156,0
EC00791=798156,0
EC00792=798156,0
EC00793=798156,0
EC00794=798156,0
EC00795=798154,1
EC00796=798154,1
EC00797=798156,0
EC00798=798156,0
EC00799=798156,0
EC00800=798156,0
EC00801=798156,0
EC00802=798156,0
EC00803=798156,0
EC00804=798156,0
EC00805=798156,0
EC00806=798156,0
EC00807=798156,0
EC00808=798156,0
EC00809=798156,0
EC00810=798156,0
EC00811=798156,0
EC00812=798156,0
EC00813=798156,0
EC00814=798156,0
EC00815=798156,0
EC00816=798156,0
EC00817=798156,0
EC00818=798156,0
EC00819=798156,0
EC00820=798156,0
EC00821=798156,0
EC00822=798156,0
EC00823=798156,0
EC00824=798156,0
EC00825=798156,0
EC00826=798156,0
EC00827=798156,0
EC00828=798156,0
EC00829=798156,0
EC00830=798156,0
EC00831=798156,0
EC00832=798156,0
EC00833=798156,0
EC00834=798156,0
EC00835=798156,0
EC00836=798156,0
EC00837=798156,0
EC00838=798156,0
EC00839=798156,0
EC00840=798156,0
EC00841=798156,0
EC00842=798156,0
EC00843=798156,0
EC00844=798156,0
EC00845=798156,0
EC00846=798156,0
EC00847=798156,0
EC00848=798156,0
EC00849=798156,0
EC00850=798156,0
EC00851=798156,0
EC00852=798156,0
EC00853=798156,0
EC00854=798156,0
EC00855=798156,0
EC00856=798156,0
EC00857=798156,0
EC00858=798156,0
EC00859=798156,0
EC00860=798156,0
EC00861=798156,0
EC00862=798156,0
EC00863=798156,0
EC00864=798156,0
EC00865=798156,0
EC00866=798156,0
EC00867=798156,0
EC00868=798156,0
EC00869=798156,0
EC00870=798156,0
EC00871=798156,0
EC00872=798156,0
EC00873=798156,0
EC00874=798156,0
EC00875=798156,0
EC00876=798156,0
EC00877=798156,0
EC00878=798156,0
EC00879=798156,0
EC00880=798156,0
EC00881=798156,0
EC00882=798156,0
EC00883=798156,0
EC00884=798156,0
EC00885=798156,0
EC00886=798156,0
EC00887=798156,0
EC00888=798156,0
EC00889=798156,0
EC00890=798156,0
EC00891=798156,0
EC00892=798156,0
EC00893=798156,0
EC00894=798156,0
EC00895=798156,0
EC00896=798156,0
EC00897=798156,0
EC00898=798156,0
EC00899=798156,0
EC00900=798156,0
EC00901=798156,0
EC00902=798156,0
EC00903=798156,0
EC00904=798156,0
EC00905=798156,0
EC00906=798156,0
EC00907=798156,0
EC00908=798156,0
EC00909=798156,0
EC00910=798156,0
EC00911=798156,0
EC00912=798156,0
EC00913=798156,0
EC00914=798156,0
EC00915=798156,0
EC00916=798156,0
EC00917=798156,0
EC00918=798156,0
EC00919=798156,0
EC00920=798156,0
EC00921=798156,0
EC00922=798156,0
EC00923=798156,0
EC00924=798156,0
EC00925=798156,0
EC00926=798156,0
EC00927=798156,0
EC00928=798156,0
EC00929=798156,0
EC00930=798156,0
EC00931=798156,0
EC00932=798156,0
EC00933=798156,0
EC00934=798156,0
EC00935=798156,0
EC00936=798156,0
EC00937=798156,0
EC00938=798156,0
EC00939=798156,0
EC00940=798156,0
EC00941=798156,0
EC00942=798156,0
EC00943=798156,0
EC00944=798156,0
EC00945=798156,0
EC00946=798156,0
EC00947=798156,0
EC00948=798156,0
EC00949=798156,0
EC00950=798156,0
EC00951=798156,0
EC00952=798156,0
EC00953=798156,0
EC00954=798156,0
EC00955=798156,0
EC00956=798156,0
EC00957=798156,0
EC00958=798156,0
EC00959=798156,0
EC00960=798156,0
EC00961=798156,0
EC00962=798156,0
EC00963=798156,0
EC00964=798156,0
EC00965=798156,0
EC00966=798156,0
EC00967=798156,0
EC00968=798156,0
EC00969=798156,0
EC00970=798156,0
EC00971=798156,0
EC00972=798156,0
EC00973=798156,0
EC00974=798156,0
EC00975=798156,0
EC00976=798156,0
EC00977=798156,0
EC00978=798156,0
EC00979=798156,0
EC00980=798156,0
EC00981=798156,0
EC00982=798156,0
EC00983=798156,0
EC00984=798156,0
EC00985=798156,0
EC00986=798156,0
EC00987=798156,0
EC00988=798156,0
EC00989=798156,0
EC00990=798156,0
EC00991=798156,0
EC00992=798156,0
EC00993=798156,0
EC00994=798156,0
EC00995=798156,0
EC00996=798156,0
EC00997=798156,0
EC00998=798156,0
EC00999=798156,0
EC01000=798156,0
EC01001=798156,0
EC01002=798156,0
EC01003=798156,0
EC01004=798156,0
EC01005=798156,0
EC01006=798156,0
EC01007=798156,0
EC01008=798156,0
EC01009=798156,0
EC01010=798156,0
EC01011=798156,0
EC01012=798156,0
EC01013=798156,0
EC01014=798156,0
EC01015=798156,0
EC01016=798156,0
EC01017=798156,0
EC01018=798156,0
EC01019=798156,0
EC01020=798156,0
EC01021=798156,0
EC01022=798156,0
EC01023=798156,0
EC01024=798156,0
EC01025=798156,0
EC01026=798156,0
EC01027=798156,0
EC01028=798156,0
EC01029=798156,0
EC01030=798156,0
EC01031=798156,0
EC01032=798156,0
EC01033=798156,0
EC01034=798156,0
EC01035=798156,0
EC01036=798156,0
EC01037=798156,0
EC01038=798156,0
EC01039=798156,0
EC01040=798156,0
EC01041=798156,0
EC01042=798156,0
EC01043=798156,0
EC01044=798156,0
EC01045=798156,0
EC01046=798156,0
///POSTYPE BASE
///RECTAN
///RCONF 0,0,0,0,0,0,0,0,0,0,0,0,0,0,0,0,0,0,0,0,0,0,0,0
P00006=0.222,-3.123,-1.508,0.0000,0.0000,0.0000
